	(* Tipologia di presa della falda *)
	TPICK_LAY_VENTOSE							:= 4,		(* Identifica la presa di tipo FALDA A VENTOSE, utilizzata nel pal. Lastre *)
	TPICK_LAY_ARPIONI							:= 5,		(* Identifica la presa di tipo FALDA CON ARPIONI, utilizzata nel pal. Lastre per il polistirolo *)
	
	TPICK_QUADROTTA								:= 10		(* Identifica la presa di tipo LASTRA (CLASSICA A VENTOSE) *)

	//TPICK_UNDEFINED								 := 99     
);
END_TYPE
//  TPICK_NOT_DEFINED = '-1'

// ---- Data types/Enum/e_Tipo_Traiettoria.TcTLEO
{attribute 'Tc2GvlVarNames'}
{attribute 'strict'}
(* Tipi Traiettoria *)
TYPE e_Tipo_Traiettoria :
(
	TRAIETTORIA_SENZA_APPROCCIO	:= 0,	(* Identifica che il punto di approccio coincide con il punto di deposito *)
	TRAIETTORIA_CON_APPROCCIO	:= 1	(* Identifica che il punto di approccio dipende dai valori di Ax,Ay,Az della lastra in deposito *)
);
END_TYPE

// ---- Data types/Enum/e_Verso_Pallettizzatore.TcTLEO
{attribute 'Tc2GvlVarNames'}
{attribute 'strict'}
//Verso del Pallettizzatore
TYPE e_Verso_Pallettizzatore :
(
	PALLETTIZZATORE_DX := 1, //Identifica il pallettizzatore la cui linea di trasporti rimane ALLE SPALLE e A DESTRA
	PALLETTIZZATORE_SX := 2 //Identifica il pallettizzatore la cui linea di trasporti rimane ALLE SPALLE e A SINISTRA
);
END_TYPE

// ---- Data types/Enum/Formatura/e_TipologiaDeposito.TcDUT
{attribute 'Tc2GvlVarNames'}
{attribute 'strict'}
TYPE e_TipologiaDeposito :
(
	NOT_DEFINED				:= -1,
	ORIZZONTALE				:= 1,		// TIPO DI DEPOSITO ORIZZONTALE (CASSA E PALLET)
	INCLINATO				:= 2,		// TIPO DI DEPOSITO INCLINATO (CAVALLINA)
	INCLINATO_LATOSINGOLO	:= 3		// TIPO DI DEPOSITO INCLINATO CON UN SOLO LATO DI DEPOSITO (BUNDLE)
);
END_TYPE

// ---- Data types/Enum/Trasporti/e_ElementZone.TcDUT
{attribute 'Tc2GvlVarNames'}
{attribute 'strict'}
TYPE e_ElementZone :
(
	NULL				:= -1,
	RullCarico 			:= 0,
	RullCarico2 		:= 1,
	RullCentrIngresso 	:= 2,
	RullCentrIngresso2 	:= 3,
	RullMobile 			:= 4,
	RullMobile2 		:= 5,
	RullP1 				:= 6,
	RullP1_2 			:= 7,
	RullP2 				:= 8,
	RullP2_2 			:= 9,
	RullSC1 			:= 10,
	RullSC1_2 			:= 11,
	RullSC2 			:= 12,
	RullSC2_2 			:= 13	
	
);
END_TYPE

// ---- Data types/Enum/Trasporti/e_PosizioneRullieraMobile.TcDUT
{attribute 'Tc2GvlVarNames'}
//{attribute 'strict'}
TYPE e_PosizioneRullieraMobile :
(
	POSIZIONE_INDEFINITA 	:= 0, 	//Posizione Indefinita
	POSIZIONE_CARICO 		:= 1,	//Posizione Rulliera Carico
	POSIZIONE_SCARICO 		:= 2,	//Posizione Rulliera Scarico
	POSIZIONE_RP1 			:= 3,	//Posizione Rulliera Prelievo 1
	POSIZIONE_RP2 			:= 4,	//Posizione Rulliera Prelievo 2
	POSIZIONE_ATTUALE 		:= 5	//Posizione Rulliera ATTUALE, NON SI CAMBIA LA DESTINAZIONE!
);
END_TYPE

// ---- Data types/Enum/Trasporti/e_StatoCentratura.TcDUT
{attribute 'Tc2GvlVarNames'}
{attribute 'strict'}
TYPE e_StatoCentratura :
(
	CENTRATURA_DISABILITATA		:= 0, 
	CENTRATURA_DA_ESEGUIRE	:= 1, 
	CENTRATURA_ESEGUITA 		:= 2
);
END_TYPE

// ---- Data types/Enum/Trasporti/e_TipoMacchinaTrasporti.TcDUT
{attribute 'Tc2GvlVarNames'}
{attribute 'strict'}
TYPE e_TipoMacchinaTrasporti :
(
	Macchina_ZonaPal := 0,//Zona Pallettizzatore
	Macchina_ZonaBS := 1 //Zona BAnco Scelta
);
END_TYPE

// ---- Data types/LGV/e_Tipo_Richiesta_LGV.TcTLEO
{attribute 'Tc2GvlVarNames'}
{attribute 'strict'}
//Tipo Richiesta LGV
TYPE e_Tipo_Richiesta_LGV :
(
	REQ_PRELIEVO_LGV_PIENO	:= 1,	(* Tipo di richiesta LGV = Richiesta di Tipo "PRELIEVO DI ELEMENTO CON MATERIALE" *)
	REQ_DEPOSITO_LGV_PIENO	:= 2,	(* Tipo di richiesta LGV = Richiesta di Tipo "DEPOSITO ELEMENTO CON MATERIALE" *)
	REQ_PRELIEVO_LGV_VUOTO	:= 3,	(* Tipo di richiesta LGV = Richiesta di Tipo "PRELIEVO ELEMENTO SENZA MATERIALE" *)
	REQ_DEPOSITO_LGV_VUOTO	:= 4	(* Tipo di richiesta LGV = Richiesta di Tipo "DEPOSITO ELEMENTO SENZA MATERIALE" *)
	
);
END_TYPE

// ---- Data types/LGV/e_Stato_Richiesta_LGV_1.TcTLEO
{attribute 'Tc2GvlVarNames'}
{attribute 'strict'}
//Stato Richiesta LGV
TYPE e_Stato_Richiesta_LGV_1 :
(
	NESSUNA_REQ_LGV	 	:= 0,	(* NESSUNA RICHIESTA/CHIAMATA LGV *)
	REQ_LGV			 	:= 1 	(* CHIAMATA LGV *)
);
END_TYPE

// ---- Data types/LGV/LGV_Stato_Formatura.TcDUT
TYPE LGV_Stato_Formatura :
STRUCT

CodicePallet 	: INT; //Codice del Pallet Presente in formatura
CodiceFalda		: INT; //Codice della Falda presente in formatura
PacchiPresenti_ZonaPositiva : INT; //Numero dei pacchi presenti della formatura nella zona Positiva(rispetto al ribaltino)
PacchiPresenti_ZonaNegativa : INT; //Numero dei pacchi presenti della formatura nella zona Negativa(rispetto al ribaltino)

END_STRUCT
END_TYPE

// ---- Data types/LGV/LGV_Stato_Pallettizzatore.TcDUT
TYPE LGV_Stato_Pallettizzatore :
STRUCT
	(* Stato del Pallettizzatore *)
	Automatico 	: BOOL; //Identifica lo stato di AUTOMATICO del Pallettizzatore
	Errore 		: BOOL; //Identifica lo stato di ERRORE del Pallettizzatore

END_STRUCT
END_TYPE

// ---- Data types/LGV/LGV_Stato_Postazione.TcDUT
TYPE LGV_Stato_Postazione :
STRUCT

	Abilitata			: INT; 	 // Abilitazione: 0=Postazione DISABILITATA, 1=Postazione ABILITATA
	Tipologia 			: INT; 	 // Tipologia: 1=Catasta Vuoti, 2=Pallet Singolo, 3=Falda,
	ProgressiveNr 		: UDINT; //Ad ogni deposito PALLET viene incrementato il suo valore ("ID univoco del pallet depositato")
	LGV_Req 			: INT; 	 //Chiamata Navetta: 0=Nessuna Chiamata, 1=Chiamata LGV
	CodicePallet 		: INT;	 //Codice identificativo del Pallet
	CodiceFalda 		: INT;	 //Codice identificativo della Falda
	CodiceLavorazione 	: INT;	 //Codice identificativo di lavorazione 
	AltezzaPallet		: REAL;	 //Altezza REALE degli elemti sulla Postazione
	
	Stato 				: INT; 	//Stato della Postazione
	CodiceFormatura 	: INT; 	//Codice di Formatura Associata alla postazione
	NPaccoSuccesivo 	: INT;	//Numero del pacco da depositare
	PN					: INT;	//Quota X postazione rispetto all quota X del ribaltino (0=Positiva, 1=Negativa)
	LGVAttr				: INT;   //Identifica gli attributi che il pallet completo dovrà avere (Tipo di Nastratura,avvolgitura,ecc)

END_STRUCT
END_TYPE

// ---- Data types/LGV/e_Stato_Operazione_LGV.TcTLEO
{attribute 'Tc2GvlVarNames'}
{attribute 'strict'}
//Stato Operazione LGV
TYPE e_Stato_Operazione_LGV :
(
	LGV_OPERAZIONE_VERIFICATA 	:= 0,	(* Indica che l'operazione svolta da parte del veicolo è stata verificata *)
	LGV_PRELIEVO_EFFETTUATO 	:= 1,	(* Indica che il prelievo da parte del veicolo è stato effettuato *)   
	LGV_DEPOSITO_EFFETTUATO 	:= 2	(* Indica che il deposito da parte del veicolo è stato effettuato *)
);
END_TYPE

// ---- Data types/Nuove/ST_OffsetAllDirection.TcDUT
TYPE ST_OffsetAllDirection :
STRUCT
	X90 : REAL := 0.0;	(* (mm) OFFSET di deposito direzione X, utilizzato per PALLET o CASSE *)
	Y90 : REAL := 0.0;	(* (mm) OFFSET di deposito direzione Y, utilizzato per PALLET o CASSE *)
	Z90 : REAL := 0.0;	(* (mm) OFFSET di deposito direzione Z, utilizzato per PALLET o CASSE *)
	J90 : REAL := 0.0;	(* (mm) OFFSET di deposito direzione J, utilizzato per PALLET o CASSE *)
	
	X0 	: REAL := 0.0;	(* (mm) OFFSET di deposito direzione X, utilizzato per CAVALLETTI *)
	Y0 	: REAL := 0.0;	(* (mm) OFFSET di deposito direzione Y, utilizzato per CAVALLETTI *)
	Z0 	: REAL := 0.0;	(* (mm) OFFSET di deposito direzione Z, utilizzato per CAVALLETTI *)
	J0 	: REAL := 0.0;	(* (mm) OFFSET di deposito direzione J, utilizzato per CAVALLETTI *)
	
	X180 : REAL := 0.0;	(* (mm) OFFSET di deposito direzione X, utilizzato per CAVALLETTI *)
	Y180 : REAL := 0.0;	(* (mm) OFFSET di deposito direzione Y, utilizzato per CAVALLETTI *)
	Z180 : REAL := 0.0;	(* (mm) OFFSET di deposito direzione Z, utilizzato per CAVALLETTI *)
	J180 : REAL := 0.0;	(* (mm) OFFSET di deposito direzione J, utilizzato per CAVALLETTI *)

END_STRUCT
END_TYPE

// ---- Data types/Nuove/TFMachinePalletizer_ListaProduzione_WAM_HMI.TcDUT
TYPE TFMachinePalletizer_ListaProduzione_WAM_HMI :
STRUCT
	Stato					: INT		:= -1;	(* Stato Elemento *)
	Support					: TFMachinePalletizer_Pallet; (* Tipologia supporto *)
	PElementList			: ARRAY [1..MAXELEMENTLIST] OF TFMachinePalletizer_PlaceElementList ; (* Elemento Da Movimentare *)
	NumeroListaAssociata 	: UINT := 0;//Indica il numero della lista associata a questa postazione nel caso ci siano + liste possibili es. post 1-4/5-8..																								
END_STRUCT
END_TYPE

// ---- Data types/Nuove/TFMachinePalletizer_WorkAreaTransport_State.TcDUT
TYPE TFMachinePalletizer_WorkAreaTransport_State :
STRUCT
	
	IDElement 		: UDINT; //ID univoco generato dalla macchina  per il tracking degli alementi
	
	State			: e_Stato_PickPoint	:= 0;	(* Stato della rulliera (0=Rulliera In Manuale, 1=Rulliera in Automatico, 2=Rulliera in Allarme *)
	PowerOK			: BOOL  := FALSE; (* Indica che ho la marcia degli ausiliari delle rulliere *)
	ProdPresence	: e_Stato_Prodotto_Generico	:= PROD_ASSENTE;	(* Stato di Presenza prodotto (0=Prodotto Assente, 1=Prodotto Presente *)
	ReadyToWork		: BOOL  := 0;	(* Indica che si puù lavorare sul supporto, quindi prelevare o depositare elementi *)
	Priority		: INT   := 0;	(* Priorità del punto di prelievo, Attualmente: 0 = Priorità MINIMA, 1 = Priorità MASSIMA *)
	
	Element			: TFMachinePalletizer_PlaceElement; (* Struttura Usata per Tracciare l'elemento presente *)
	DataElement		: TFMachinePalletizer_DataElement; (* Struttura dati che la macchina acquisisce/trasferisce in fase di pallettizzazione/depallettizazione *)
	Supporto		: TFMachinePalletizer_Pallet; (* Struttura del supporto presente sul punto di prelievo *)
	
	StatoPrelievo	: INT   := 0;	(* WRITE - Stato del prelievo: 0 = Da effettuare, 1 = Effettuato *)		
	StatoIngombroEE	: INT   := 0;	(* WRITE - Stato dell'ingombro dell'End-Effector: 0 = Non in ingombro, 1 = In Ingombro *)	
	
	XPosBandella		: REAL  := 0.0; (* Quota Bandella, Scritta dalle Rulliere (se posizionamento motorizzato) oppure dall'operatore (misura dal punto fiso della rulliera alla bandella) *)
	YPosBandella		: REAL  := 0.0; (* Quota Bandella, Scritta dalle Rulliere (se posizionamento motorizzato) oppure dall'operatore (misura dal punto fiso della rulliera alla bandella) *)
	
	NumeroPrelDepEffettuati : UINT := 0; (* Numero prelievi/Depositi effettuati sulle'elemento attuale *)
	
END_STRUCT
END_TYPE

// ---- Data types/Nuove/TFMachinePalletizer_WorkPlacePointToPalletizer.TcDUT
TYPE TFMachinePalletizer_WorkPlacePointToPalletizer :
STRUCT

	State					: e_Stato_PickPoint	:= 0;	(* Stato della rulliera (0=Rulliera In Manuale, 1=Rulliera in Automatico, 2=Rulliera in Allarme *)
                         
	PhaseStopDone 			: BOOL;(*Richiesta Stop in fase ESEGUITA*)
                            
	IDElement 				: UDINT; (*ID univoco generato dalla macchina  per il tracking degli alementi*)
	SupportPresent 		 	: BOOL;(* Supporto presente sul punto di deposito e pronto per essere pallettizzato *) 	
	Support 				: TFMachinePalletizer_Pallet; (* Struttura del supporto presente sul punto di prelievo *)
		
END_STRUCT
END_TYPE

// ---- Data types/Nuove/TFMachinePalletizer_WorkPlacePointFromPalletizer.TcDUT
TYPE TFMachinePalletizer_WorkPlacePointFromPalletizer :
STRUCT

	PhaseStopReq 			: BOOL;(*Richiesta Stop in fase*)
                            
	SupportREQ 				: BOOL;(* Richiesta del supporto punto di depostio *)
	Support				  	: TFMachinePalletizer_Pallet;(* Struttura del supporto richiesto sul punto di deposito *)
                                                 
	StatoIngombroEE			: INT   := 0;	(* Stato dell'ingombro dell'End-Effector: 0 = Non in ingombro, 1 = In Ingombro *)	
	
	ElementCompleted		: BOOL; (* Indica che l'elemento è stato completato *)

	State					: INT;//STtao pallettizzatore

	NextSupport			  	: TFMachinePalletizer_Pallet;(* Struttura del supporto successivo richiesto sul punto di deposito *)
   
END_STRUCT
END_TYPE

// ---- Data types/Picking/e_TypologySupDataPicking.TcDUT
{attribute 'strict'}
TYPE e_TypologySupDataPicking :
(
	//0= Orrizzontale LEGNO,1= Orrizzontale Telaio , 2 = Bundle, 3 = A-FRAME
	LEGNO_PIANO 	:= 0, //Legno/Pallet in piano
	TELAIO_PIANO 	:= 1, //Telaio in ferro in piano
	BUNDLE_VERT 			:= 2, //Bundle posteriore
	A_FRAME_VERT 		:= 3 //A-FRAME 
);
END_TYPE

// ---- Data types/Picking/ST_DataManualPicking.TcDUT
TYPE ST_DataManualPicking :
STRUCT
	ID_LIST			: STRING(255) 	:= '';	(* Identificatore univoco della LISTA da Eseguire *)
	State			: INT			:= -1;	(*Stato della lista in lavoro *)
	SlabNumber  	: UINT 			:= 0; (* Numero di lastre da depositare sul supporto *)
	SlabDimension 	: TFDimensionElement; (* Dimensione Lastra *)
	Layer 			: ST_LayerData; (* Struttura descrizione falda *)
	LayerSequence 	: INT; (* Sequenza di deposito delle falde -> 0=Nessuna falda,1=Deposito dopo ogni lastra,2=Deposito ogni 2 lastre,ecc*)
	SupportPianoLegno	: ST_SupportData; (* Dati del supporto in piano per legni*)
	SupportPianoFerro	: ST_SupportData; (* Dati del supporto in piano per ferro*)
	SupportVertBundle	: ST_SupportData; (* Dati del supporto in verticale per bundle*)	
	SupportVertCav		: ST_SupportData; (* Dati del supporto in verticale per cavalletto*)	
END_STRUCT
END_TYPE

// ---- Data types/Picking/ST_WorkAreaDataPicking.TcDUT
TYPE ST_WorkAreaDataPicking :
STRUCT
	Destinazione		  		: BOOL;	//Se TRUE=WA di destinazione materiale, FALSE=Postazione di prelievo materiale
	NumElementiDaLavorare 		: UINT; 	//Numero elementi da depositare-prelevare
	Typology			  		: INT := 0; 	//Supporto disposto in verticale: e_TypologySupDataPicking: 0= Orrizzontale LEGNO,1= Orrizzontale Telaio , 2 = Bundle, 3 = A-FRAME 
	TipoTrabajoLado_Cavallete 	: INT := 0; // // 0-trabaja aambos lados 1-Lado 0 Grados 2-Lado 180 Grados
END_STRUCT
END_TYPE

// ---- Data types/Programmi Movimento/TFModulePortaleStatus.TcDUT
TYPE TFModulePortaleStatus :
STRUCT
	
	X				: ST_MachinePalletizerAxeState;	(* X Axe State (UI Position=mm, UI Velocity=mm/sec UI Acc/Dec=mm/sec2) *)
	Y				: ST_MachinePalletizerAxeState;	(* Y Axe State (UI Position=mm, UI Velocity=mm/sec UI Acc/Dec=mm/sec2) *)
	Z				: ST_MachinePalletizerAxeState;	(* Z Axe State (UI Position=mm, UI Velocity=mm/sec UI Acc/Dec=mm/sec2) *)
	J				: ST_MachinePalletizerAxeState;	(* J Axe State (UI Position=°,  UI Velocity=°/sec  UI Acc/Dec=°/sec2) *)
	K				: ST_MachinePalletizerAxeState;	(* K Axe State (UI Position=mm, UI Velocity=mm/sec UI Acc/Dec=mm/sec2) *)
	Pinza 			: ST_MachinePalletizerPinzaStateComplete; (* State Pinza *)
	
	Macchina   		: ST_MachinePalletizerMachineState; (* Stato del modulo di gestione Della Macchina *)

	ModAsse_X 		: ST_MachinePalletizerModuleState; (* Stato del modulo di gestione Asse X *)
	ModAsse_Y 		: ST_MachinePalletizerModuleState; (* Stato del modulo di gestione Asse Y *)
	ModAsse_Z 		: ST_MachinePalletizerModuleState; (* Stato del modulo di gestione Asse Z *)
	ModAsse_J 		: ST_MachinePalletizerModuleState; (* Stato del modulo di gestione Asse J *)
	ModAsse_K 		: ST_MachinePalletizerModuleState; (* Stato del modulo di gestione Asse K *)
	ModPinza 		: ST_MachinePalletizerModuleState; (* Stato del modulo di gestione Pinza *)
	ModLettoreBc 	: ST_MachinePalletizerModuleState; (* Stato del modulo di gestione Lettore Barcode *)
	
END_STRUCT
END_TYPE

// ---- Data types/StatoPostazioneHMI.TcDUT
TYPE StatoPostazioneHMI :
STRUCT

	Abilitata			: INT; 	 // Abilitazione: 0=Postazione DISABILITATA, 1=Postazione ABILITATA
	TipologiaPostazione	: INT; 	 // Tipologia: 1=Catasta Vuoti, 2=Pallet Singolo, 3=Falda,
	ProgressiveNr 		: UDINT; //Ad ogni deposito PALLET viene incrementato il suo valore ("ID univoco del pallet depositato")
	
	LGV_Req 			: INT; 	 //Chiamata Navetta: 0=Nessuna Chiamata, 1=Chiamata LGV
	TipologiaSupporto   : INT;
	CodiceLavorazione 	: INT;	 //Codice identificativo di lavorazione 
	
	Stato 				: INT; 	//Stato della Postazione
	CodiceFormatura 	: INT; 	//Codice di Formatura Associata alla postazione
	NPezzi			 	: INT;	//Numero dei pezzi presenti
	

END_STRUCT
END_TYPE

// ---- Data types/Nuove/TFCodiciPerFormatura.TcDUT
TYPE TFCodiciPerFormatura :
STRUCT
	Code : ARRAY[1..MAXFORMINGCODE] OF INT;
END_STRUCT
END_TYPE

// ---- Data types/Nuove/TFError_WAM.TcDUT
TYPE TFError_WAM :
STRUCT
	Code 		: UINT; (*Codice di errore*)
	ExtraCode 	: UINT; (*Codice di errore EXTRA*)
END_STRUCT
END_TYPE

// ---- Data types/Nuove/TFMachinePalletizer_DataElementMP.TcDUT
TYPE TFMachinePalletizer_DataElementMP :
STRUCT
	RequetsID 		: DINT	:= 0; (* Scheduler ID *)
	Article 			: STRING(49) := '';
	ArticleDescription 	: STRING(49) := '';(* Descrizione Articolo *)
	Tono			: STRING(19)	:= '';	(* Tono Elemento *)
	Scelta			: STRING(19)	:= '';	(* Scelta Elemento *)
	Calibro			: STRING(19)	:= '';	(* Calibro Elemento *)
	
	Lenght 		: INT := 0; //Lunghezza
	Width 		: INT := 0; //Larghezza
	Thickness 	: INT := 0; //Spessore
END_STRUCT
END_TYPE

// ---- Data types/Nuove/TFMachinePalletizer_PinzaVentoseManCmd.TcDUT
TYPE TFMachinePalletizer_PinzaVentoseManCmd :
STRUCT
	
	AttivazioneVuotoDX			: BOOL;//Attivazione vuoto Ovem DX 
	AttivazioneVuotoSX			: BOOL;//Attivazione vuoto Ovem SX

	DisattivazioneVuotoDX			: BOOL;//Comandi Ovem
	DisattivazioneVuotoSX			: BOOL;//Comandi Ove

	ApriPinza				: BOOL; //Apertura Pinza
	ChiudiPinza				: BOOL; //Apertura Pinza

	SbloccoPinza			: BOOL;//Sblocco rotazione
	BloccoPinza				: BOOL;//Blocco rotazione

	AttivazioneVuotoFaldeDX 	: BOOL;//Attivazione aspirazione Falde DX
	DisattivazioneVuotoFaldeDX	: BOOL;//Disattivazione aspirazione Falde DX
	
	AttivazioneVuotoFaldeSX 	: BOOL;//Attivazione aspirazione Falde SX
	DisattivazioneVuotoFaldeSX	: BOOL;//Disattivazione aspirazione Falde SX

	AttivaTastatori : BOOL; //Attivazione Tastatori
	DisattivaTastatori : BOOL; //Disattivazione Tastatori
	
	CalibrazioneOVEM : bool; //Calibrazione OVEM

END_STRUCT
END_TYPE

// ---- Data types/Nuove/TFMachinePalletizer_ApprendimentoQuota.TcDUT
TYPE TFMachinePalletizer_ApprendimentoQuota :
STRUCT
	Stato			: e_Stato_Apprendimento	:= e_Stato_Apprendimento.NOT_DEFINED;	(* Stato apprendimento Direzione X 0=Disabilitato, 1=Abilitato da Eseguire, 2=Eseguito, -1 dato non valido *)
	QuotaStart		: LREAL	:= 0.0;	(* (mm) Quota inizio Apprendimento Direzione X *)
	QuotaRilevata	: LREAL	:= 0.0; (* Quota rilevata durante apprendimento Direzione X *)
END_STRUCT
END_TYPE

// ---- Data types/Nuove/TFMachinePalletizer_CoordinateApprendimento.TcDUT
TYPE TFMachinePalletizer_CoordinateApprendimento :
STRUCT
	X : TFMachinePalletizer_LatoApprendimento;
	Y : TFMachinePalletizer_LatoApprendimento;
	Z : TFMachinePalletizer_LatoApprendimento;
	J : TFMachinePalletizer_LatoApprendimento;
END_STRUCT
END_TYPE

// ---- Data types/Nuove/TFMachinePalletizer_LatoApprendimento.TcDUT
TYPE TFMachinePalletizer_LatoApprendimento :
STRUCT
	Lato0 	: TFMachinePalletizer_ApprendimentoQuota;	
	Lato90 	: TFMachinePalletizer_ApprendimentoQuota;
	Lato180 : TFMachinePalletizer_ApprendimentoQuota;
END_STRUCT
END_TYPE

// ---- Data types/Nuove/TFMachinePalletizer_DataElement.TcDUT
TYPE TFMachinePalletizer_DataElement :
STRUCT
	WorkingID 			: STRING	:= ''; (* Identifica l'ID univoco della lavorazione da eseguire *)
	
	Codice				: STRING	:= '';	(* Codice Elemento *)
	Scelta				: STRING	:= '';	(* Scelta Elemento *)
	Tono				: STRING	:= '';	(* Tono Elemento *)
	Calibro				: STRING	:= '';	(* Calibro Elemento *)
	Quantity  			: UINT 		:= 0;	(* Quantità *)
	ArticleDescription 	: STRING(50) := '';(* Descrizione Articolo *)
END_STRUCT
END_TYPE

// ---- Data types/Nuove/TFMachinePalletizer_EndEffector.TcDUT
TYPE TFMachinePalletizer_EndEffector :
STRUCT
	Tipologia 	: INT := -1; 	//Indica la tipologia dell'elemento 
	Lunghezza 	: REAL := 0; 	//Indica la lunghezza dell'elemento
	Larghezza 	: REAL := 0; 	//Indica la larghezza dell'elemento	
	Spessore	: REAL := 0; 	//Indica lo spessore dell'elemento
	PosizioneBC_X : REAL := 0;	//Indica la posizione del barcode lungo la sua lunghezza e rispetto il punto medio
	PosizioneBC_Y : REAL := 0;	//Indica la posizione del barcode lungo la sua larghezza e rispetto il punto medio	
	PosizioneBC_Z : REAL := 0;	//Indica la posizione del barcode lungo il suo spessore e rispetto il punto medio
END_STRUCT
END_TYPE

// ---- Data types/Nuove/TFMachinePalletizer_BarCode.TcDUT
TYPE TFMachinePalletizer_BarCode :
STRUCT
	State 	: e_Stato_LetturaBarCode := LETURA_BC_TERMINATA;				(* Identifica lo stato della Lettura del BC:	0= Non Ancora letto/Da Leggere, 
																					1= Lettura In corso
																					2= Codice Letto e Valido/Non da leggere, 
																					3= Errore *)
	ErrorCode	: INT := 0;				(* Identifica il codice di errore *)
	Value		: STRING[DIMBARCODE];	(* Identifica il valore della lettura *)	
END_STRUCT
END_TYPE

// ---- Data types/Nuove/TFMachinePalletizer_ListaProduzione.TcDUT
TYPE TFMachinePalletizer_ListaProduzione :
STRUCT
	ID_LIST		: STRING(255) 					:= '';	(* Identificatore univoco della LISTA da Eseguire *)
	State		: e_Stato_ListaDiProduzione		:= -1;	(*Stato della lista in lavoro *)
	SlabNumber  : UINT := 0; (* Numero di lastre da depositare sul supporto *)
	SlabData 	: ARRAY[1..MAXARTICLEPICKING] OF TFMachinePalletizer_DataElement; (* Lastra che serve per comporre l'ordine finale, ordinato in base alla sequenza richiesta 1=Primo prodotto da pallettizzare *)
	SlabDimension 	: TFDimensionElement; (* Dimensione Lastra *)
	LayerSequence 	: UINT := 0;//Sequenza di deposito delle falde -> 0=Nessuna falda,1=Deposito dopo ogni lastra,2=Deposito ogni 2 lastre,ecc
	LayerCode     	: UDINT := 0; (* Codice della falda da deposotare *)
	Support			: UDINT := 0; (* Codice pallet su cui eseguire la pallettizzazione *)
											
END_STRUCT
END_TYPE

// ---- Data types/Nuove/TFMachinePalletizer_ListaProduzione_WAM.TcDUT
TYPE TFMachinePalletizer_ListaProduzione_WAM :
STRUCT
	Stato					: e_Stato_ListaDiProduzione		:= -1;	(* Stato Elemento *)
	Support					: TFMachinePalletizer_Pallet; (* Tipologia supporto *)
	PElementList			: ARRAY [1..MAXELEMENTLIST] OF TFMachinePalletizer_PlaceElementList ; (* Elemento Da Movimentare *)
	Forming 				: TFMachinePalletizer_FormingForSlab;
	NumeroListaAssociata 	: UINT := 0;//Indica il numero della lista associata a questa postazione nel caso ci siano + liste possibili es. post 1-4/5-8..												
END_STRUCT
END_TYPE

// ---- Data types/Nuove/TFMachinePalletizer_OffsetElement.TcDUT
TYPE TFMachinePalletizer_OffsetElement :
STRUCT
	Dir_X 				: REAL := 0.0;	(* (mm) OFFSET in direzione X *)
	Dir_Y 				: REAL := 0.0;	(* (mm) OFFSET in direzione Y (+ è grande + mi allontano dal supporto)*)
	Dir_Z 				: REAL := 0.0;	(* (mm) OFFSET in direzione Z (+ è grande + mi allontano dal supporto)*)
	Dir_J 				: REAL := 0.0;	(* (°) OFFSET di inclinazione J (Pinza Inclinata: + è grande + è grande l'inclinazione, 
																		Pinza Pari: più è grande più si sposta verso l'angolo maggiore *)
	
END_STRUCT
END_TYPE

// ---- Data types/Nuove/TFMachinePalletizer_PickPlaceParameters.TcDUT
TYPE TFMachinePalletizer_PickPlaceParameters :
STRUCT

	OffsetZPlaceLayer			: REAL;	(* Offset quota Z per rilascio falda *)
			
	XPickApproach	: LREAL	:= 100.0;		(* (mm) Offset di Approccio X in prelievo *)
	YPickApproach	: LREAL	:= 100.0;		(* (mm) Offset di Approccio Y in prelievo *)
	ZPickApproach	: LREAL	:= 100.0;		(* (mm) Offset di Approccio Z in prelievo *)
	JPickApproach	: LREAL	:= 100.0;		(* (mm) Offset di Approccio J in prelievo *)
	//KPickApproach	: LREAL	:= 0.0;		(* (mm) Offset di Approccio in prelievo *)
	//WPickApproach	: LREAL	:= 0.0;		(* (mm) Offset di Approccio in prelievo *)
	
	XPlaceApproach	: LREAL	:= 100.0;		(* (mm) Offset di Approccio X in deposito *)
	YPlaceApproach	: LREAL	:= 100.0;		(* (mm) Offset di Approccio Y in deposito *)
	ZPlaceApproach	: LREAL	:= 100.0;		(* (mm) Offset di Approccio Z in deposito *)
	JPlaceApproach	: LREAL	:= 100.0;		(* (mm) Offset di Approccio in deposito *)
	//KPlaceApproach	: LREAL	:= 0.0;		(* (mm) Punto di Approccio in deposito *)
	//WPlaceApproach	: LREAL	:= 0.0;		(* (mm) Punto di Approccio in deposito  *)

END_STRUCT
END_TYPE

// ---- Data types/Nuove/TFMachinePalletizer_PinzaState.TcDUT
TYPE TFMachinePalletizer_PinzaState :
STRUCT
	LatoDxAperto : BOOL; //Indica che la prolunga DX della pinza è aperta
	LatoSxAperto : BOOL; //Indica che la prolunga SX della pinza è aperta
	LatoDxChiuso : BOOL; //Indica che la prolunga DX della pinza è chiusa
	LatoSxChiuso : BOOL; //Indica che la prolunga SX della pinza è chiusa
	
	LatoSxPiastrellaInPresa : BOOL; //Indica che sul lato SX ho in presa la piastrella
	LatoDxPiastrellaInPresa : BOOL; //Indica che sul lato DX ho in presa la piastrella

	LatoSxFaldaInPresa 		: BOOL; //Indica che sul lato SX ho in presa la FALDA
	LatoDxFaldaInPresa 		: BOOL; //Indica che sul lato DX ho in presa la FALDA
	
	RotazioneSbloccata 	: BOOL; //Indica che la Rotazione lungo z è sbloccata
	RotazioneBloccata	: BOOL; //Indica che la rotazione lungo z è bloccata
	
	ElementoPrelevato : BOOL;//Indica che l'elemento è stato prelevato
	
	LetturaFTC0 	: REAL;
	LetturaFTC180 	: REAL;
	
	LetturaFTC0_2 	: REAL;
	LetturaFTC180_2 : REAL;
	
	PianoInPresa : BOOL;
END_STRUCT
END_TYPE

// ---- Data types/Nuove/TFMAchinePalletizer_PinzaVentoseStatus.TcDUT
TYPE TFMAchinePalletizer_PinzaVentoseStatus :
STRUCT

	Module : TFMachinePalletizer_ModuleState;

	CilindroApertura 			: TF_CylinderState;
	CilindroSbloccoRotazione 	: TF_CylinderState;
	AspirazioneFaldaDX 			: TF_CylinderState;
	AspirazioneFaldaSX 			: TF_CylinderState;
	AspirazioneDX 				: TF_CylinderState;
	AspirazioneSX 				: TF_CylinderState;		
	CilindroTasteggio			: TF_CylinderState;	
	AspirazioneDX2 				: TF_CylinderState;
	AspirazioneSX2 				: TF_CylinderState;		
	CilindroSbloccoBascolante 	: TF_CylinderState;
END_STRUCT
END_TYPE

// ---- Data types/Nuove/TFMachinePalletizer_PinzaVentose_OUT.TcDUT
TYPE TFMachinePalletizer_PinzaVentose_OUT :
STRUCT
END_STRUCT
END_TYPE

// ---- Data types/Nuove/TFMachinePalletizer_PlaceElement.TcDUT
TYPE TFMachinePalletizer_PlaceElement :
STRUCT
	(* Tipologia *)
	Typology		: e_Tipo_Elemento_Da_Lavorare := TERMINATORE;	(* Tipo di ELEMENTO DA LAVORARE: 0: LASTRA,1:FALDA *)
	TypologyCode	: INT						:= -1;	(* Descrittore tipo elemento *)
	(*Dimensione Lastra*) // Añadido Alberto 14-10-2025
	SlabDimension 								: TFDimensionElement; (* Dimensione Lastra *)
	DimensionPiezasLadoALadoB					: ES_dimensionPiezaLadoA_ladoB; 
	(* Dimensioni *)
	XDim		: REAL							:= 0.0;	(* (mm) Dimensione X *)
	YDim		: REAL							:= 0.0;	(* (mm) Dimensione Y *)
	ZDim		: REAL							:= 0.0;	(* (mm) Dimensione Z *)
	(* Quote di deposito *)
	X			: LREAL							:= 0.0;	(* (mm) Destination - Coordinata X *)
	Y			: LREAL							:= 0.0;	(* (mm) Destination - Coordinata Y *)
	Z			: LREAL							:= 0.0;	(* (mm) Destination - Coordinata Z *)
	J			: LREAL							:= 0.0;	(* (°)  Destination - Coordinata J (PITCH)*)
	CooCavallete : Es_CoordenadasCaballeteLadoA_ladoB  ;
	//K			: LREAL							:= 0.0;	(* (°)  Destination - Coordinata K (ROLL)*)
	//W			: LREAL							:= 0.0;	(* (°)  Destination - Coordinata W (YAW)*)

	(* Distanza di Accostamento *)
	AX			: REAL							:= 0.0; (* (mm) Approach X Distance - Distanza Accostamento X *)
	AY			: REAL							:= 0.0; (* (mm) Approach Y Distance - Distanza Accostamento Y *)
	AZ			: REAL							:= 0.0; (* (mm) Approach Z Distance - Distanza Accostamento Z *)
	AJ			: REAL							:= 0.0; (* (mm) Approach J Distance - Distanza Accostamento J (PITCH)*)
	//NUOVE???
	//AK			: REAL						:= 0.0; (* (mm) Approach Z Distance - Distanza Accostamento K (ROLL)*)
	//AW			: REAL						:= 0.0; (* (mm) Approach J Distance - Distanza Accostamento W (YAW)*)
	(* traiettoria di deposito *)
	Trajectory	: e_Tipo_Traiettoria			:= 0;	(* READ	- Tipo di percorso (0, 1, 2, 3, …) (-1 dato non valido) *)
	Empty : BOOL;//Indica che è vuoto
END_STRUCT
END_TYPE

// ---- Data types/Nuove/TFMachinePalletizer_PlaceElementList.TcDUT
TYPE TFMachinePalletizer_PlaceElementList :
STRUCT
	
	Stato 			: e_Stato_ElementoLista; (* Stato dell'elemento della lista*)
	
	PElement 		: TFMachinePalletizer_PlaceElement; (* Elemento Da Movimentare *)
	SlabData     	: TFMachinePalletizer_DataElement; (* Dati Elemento da depositare*)

	WA_PRELIEVO		: UINT	:= 0;	(* WA DOVE VIENE FATTO IL PRELIEVO *)
	WA_DEPOSITO		: UINT	:= 0;	(* WA DOVE VIENE FATTO IL DEPOSITO *)
	PP_PRELIEVO     : UINT	:= 0;	(* PICK-POINT DOVE VIENE FATTO IL PRELIEVO *)	
	
	Pareggiatura    : e_Stato_Pareggiatura_Lastra  := PAREGGIATURA_DISABILITATA;	(* Pareggiatura Lastra da eseguire Prima del deposito 0:NON ESEGUIRE, 1: DA ESEGUIRE, 2:ESEGUITA *)
	
END_STRUCT
END_TYPE

// ---- Data types/Nuove/TFMachinePalletizer_WorkPickPointOffset.TcDUT
TYPE TFMachinePalletizer_WorkPickPointOffset :
STRUCT
	X	:	REAL := 0.0; (* READ	- (mm) Offset del punto di prelievo in direzione X *)
	Y	:	REAL := 0.0; (* READ	- (mm) Offset del punto di prelievo in direzione Y *)
	Z	:	REAL := 0.0; (* READ	- (mm) Offset del punto di prelievo in direzione Z *)
	J	:	REAL := 0.0; (* READ	- (mm) Offset di rotazione del piano J *)
END_STRUCT
END_TYPE

// ---- Data types/Nuove/TFMachinePalletizer_WorkPickPoint_State.TcDUT
TYPE TFMachinePalletizer_WorkPickPoint_State :
STRUCT
	
	State			: INT	:= 0;	(* Stato della rulliera (0=Rulliera In Manuale, 1=Rulliera in Automatico, 2=Rulliera in Allarme *)
	PowerOK			: BOOL  := FALSE; (* Indica che ho la marcia degli ausiliari delle rulliere *)
	ProdPresence	: INT	:= 0;	(* Stato di Presenza prodotto (0=Prodotto Assente, 1=Prodotto Presente *)
	LastraPronta	: BOOL  := 0;	(* Indica che la lastra è pronta per essere prelevata *)
	Code			: INT	:= 0;	(* Codice Elemento *)
	Priority		: INT   := 0;	(* Priorità del punto di prelievo, Attualmente: 0 = Priorità MINIMA, 1 = Priorità MASSIMA *)
	
	Element			: TFMachinePalletizer_PlaceElement; (* Struttura Usata per Tracciare l'elemento presente *)

	StatoPrelievo	: INT   := 0;	(* WRITE - Stato del prelievo: 0 = Da effettuare, 1 = Effettuato *)		
	StatoIngombroEE	: INT   := 0;	(* WRITE - Stato dell'ingombro dell'End-Effector: 0 = Non in ingombro, 1 = In Ingombro *)	
	
	XPosBandella		: REAL  := 0.0; (* Quota Bandella, Scritta dalle Rulliere (se posizionamento motorizzato) oppure dall'operatore (misura dal punto fiso della rulliera alla bandella) *)
	YPosBandella		: REAL  := 0.0; (* Quota Bandella, Scritta dalle Rulliere (se posizionamento motorizzato) oppure dall'operatore (misura dal punto fiso della rulliera alla bandella) *)
	
	DataElement		: TFMachinePalletizer_DataElement; (* Struttura dati che la macchina acquisisce/trasferisce in fase di pallettizzazione/depallettizazione *)
		
END_STRUCT
END_TYPE

// ---- Data types/Nuove/TFMachinePalletizer_WorkPickPointRoller_State_DaLinea.TcDUT
TYPE TFMachinePalletizer_WorkPickPointRoller_State_DaLinea :
STRUCT
	
	Automatico		: BOOL	:= FALSE;	(* Stato della rulliera (FALSE=Rulliera In Manuale, TRUE=Rulliera in Automatico *)
	Errore			: BOOL	:= FALSE;	(* Stato della rulliera (FALSE=Rulliera senza Errori, TRUE=Rulliera in Errore *)
	PowerOK			: BOOL	:= FALSE;	(* Presenza Marcia (FALSE=Marcia Assente, TRUE=Marcia Presente *)
	Codice			: INT	:= 0;		(* Codice Prodotto *)
	Occupato		: BOOL  := FALSE;	(* Rulliera Occupata *)
	LastraPronta	: BOOL  := FALSE;	(* Lastra pronta e in posizione per prelievo *)
	Priority		: BOOL	:= FALSE;	(* Se true a parità di occupazione rispetto agli altri PickPoint, questo PickPoint ha la precedenza nel prelievo *)
	
END_STRUCT
END_TYPE

// ---- Data types/Nuove/TFMachinePalletizer_WorkPickPointRoller_State_ALinea.TcDUT
TYPE TFMachinePalletizer_WorkPickPointRoller_State_ALinea :
STRUCT
	
	Automatico			: BOOL 	:= FALSE;	(* Stato della rulliera (FALSE=Rulliera In Manuale, TRUE=Rulliera in Automatico *)
	PowerOK				: BOOL 	:= FALSE; 	(* Presenza Marcia (FALSE=Marcia Assente, TRUE=Marcia Presente *)
	Ingombro			: BOOL	:= FALSE;	(* Stato della rulliera (FALSE=Rulliera In Manuale, TRUE=Rulliera in Automatico *)
	Prelievo_Effettuato	: BOOL	:= FALSE ;	(* Se TRUE il prelievo è stato effettuato *)
	
END_STRUCT
END_TYPE

// ---- Data types/Nuove/TFMachinePalletizer_WorkPickPointStore_State.TcDUT
TYPE TFMachinePalletizer_WorkPickPointStore_State :
STRUCT
	
	ProdPresence	: INT	:= 0;	(* Stato PickPoint (0=Prodotto Assente, 1=Prodotto Presente *)
	Code			: INT   := -1;	(* Indica il codice della falda *)
		
	XDim			: REAL	:= 0;		(* (mm) Dimensione X Prodotto *)
	YDim			: REAL	:= 0;		(* (mm) Dimensione Y Prodotto *)
	ZDim			: REAL	:= 0;		(* (mm) Dimensione Z Prodotto *)
	
END_STRUCT
END_TYPE

// ---- Data types/Nuove/TFMachinePalletizer_WorkPickPointSlab.TcDUT
TYPE TFMachinePalletizer_WorkPickPointSlab :
STRUCT
	
	Tipologia			: e_Tipo_PickPoint 	:= -1;		(* Tipologia del punto di prelievo 
														Per lastre 	= RULLIERA;
														Per Falde	= MAGAZZIONO_FALDE *)
														
	ID					: INT 	:= -1;		(* Identifica il numero del PickPoint *)
	Enable				: INT	:= -1;		(* PickPoint Abilitata 0=no, 1=si, -1 dato non valido *)	
(***********************************************************************************************************************************************)
	X					: LREAL	:= 0.0;		(* (mm) Quota assoluta di impianto DA ORIGINE *)
	Y					: LREAL	:= 0.0;		(* (mm) Quota assoluta di impianto DA ORIGINE *)
	Z					: LREAL	:= 0.0;		(* (mm) Quota assoluta di impianto DA ORIGINE Caso di magazzino falde: è la quota della base di appoggio*)
	J					: LREAL	:= 0.0;		(* (mm) Quota assoluta di impianto DA ORIGINE *)
	ZRaise				: REAL  := 0.0; 	(* (mm) Quota di salita per uscire dall'ingombro *)
	
	///Lunghezza			: REAL := 0.0;		(* (mm) Ingombro in Lunghezza "X" rispetto il suo centro *)
	//Larghezza			: REAL := 0.0;		(* (mm) Ingombro in Larghezza "Y" rispetto il suo centro *)
	//Altezza				: REAL := 0.0;		(* (mm) Ingombro in Altezza "Z" rispetto il suo centro *)
	
	DoLearn_Z			: e_Stato_Apprendimento	:= -1;	(* Stato apprendimento Direzione Z 0=Disabilitato, 1=Abilitato da Eseguire, 2=Eseguito, -1 dato non valido *)
	Learn_Z				: REAL	:= 0.0;	(* (mm) Quota inizio Apprendimento Direzione Z *)
	Learned_Z			: LREAL	:= 0.0; (* (mm) Quota rilevata durante apprendimento Direzione Z *)
			
END_STRUCT
END_TYPE

// ---- Data types/Nuove/TF_CylinderState.TcDUT
TYPE TF_CylinderState :
STRUCT
	Active : BOOL;
	Inactive : BOOL;
	Error : UDINT;
	SensorActive : BOOL;
	SensorInactive : BOOL;
	StatusToHMI	: uint; //0= Null; 1= Active ; 2= Inactive; 3= Idle; 9 = Error ; 
END_STRUCT
END_TYPE

// ---- Data types/Nuove/TFMchinePalletizer_PinzaVentose_IN.TcDUT
TYPE TFMchinePalletizer_PinzaVentose_IN :
STRUCT
	TastoreCartoneSX : BOOL; //Sensore Tastatore lato SX
	TastoreCartoneDX : BOOL; //Sensore Tastatore lato SX
	ExtraCorsaPinzaSganciata : BOOL; //Sensore Di sicurezza rotazione lungo Z
	
	InKeyence0_Byte0 : BYTE;
	InKeyence0_Byte1 : BYTE;
	InKeyence180_Byte0 : BYTE;
	InKeyence180_Byte1 : BYTE;
	
	InKeyence0_Byte0_2 : BYTE;
	InKeyence0_Byte1_2 : BYTE;
	InKeyence180_Byte0_2 : BYTE;
	InKeyence180_Byte1_2 : BYTE;

	ByPassSensoreVuoto : BOOL;
	RichiestaRicalibrazioneOvemEsterna : BOOL;//Richiesta calibrazione esterna da macchina
	
	FTC_FaldaDX : BOOL;
	FTC_FaldaSX : BOOL;
	
END_STRUCT
END_TYPE

// ---- Data types/Nuove/TFPalletizerModules.TcDUT
TYPE TFPalletizerModules :
STRUCT
	AX_X 	: TFModulePalletizer_Ax;
	AX_Y 	: TFModulePalletizer_Ax;
	AX_Z 	: TFModulePalletizer_Ax;
	//AX_K 	: TFModulePalletizer_Ax;
	AX_J 	: TFModulePalletizer_AxJ_Lastre;
	Pinza 	: TFModulePalletizer_Pinza;
	

END_STRUCT
END_TYPE

// ---- Data types/Programmi Movimento/AxHomingParameters.TcDUT
TYPE AxHomingParameters :
STRUCT
	TipoHoming : INT; //Tipologia di homing da eseguire
	InvertiDirezione : BOOL; //FALSE=Direzione NEgativa, TRUE=Direzione positiva
END_STRUCT
END_TYPE

// ---- Data types/Programmi Movimento/Ax_Palletizer_Basic_Parameters.TcDUT
TYPE Ax_Palletizer_Basic_Parameters :
STRUCT
	Vel 	: REAL;
	Acc 	: REAL;
	Dec 	: REAL;
	Jerk 	: REAL;
	Torque 	: REAL;
END_STRUCT
END_TYPE

// ---- Data types/Programmi Movimento/Ax_Palletizer_Nominal_Parameters.TcDUT
TYPE Ax_Palletizer_Nominal_Parameters :
STRUCT
	ReferenceVelocity 		: REAL := 0.0;
	MaximumAcceleration 	: REAL := 0.0;
	MaximumDeceleration 	: REAL := 0.0;
	DefaultJerk 			: REAL := 0.0;
	DefaultTorque 			: REAL := 100.0;
END_STRUCT
END_TYPE

// ---- Data types/Programmi Movimento/Enum Programmi/e_ProgrammiMovimentoX.TcTLEO
{attribute 'Tc2GvlVarNames'}
{attribute 'strict'}
TYPE e_ProgrammiMovimentoX :
(
	
	X_PosDiRiposo					:= 0,
	X_PosFuoriIngombroRiposo 			:= 6,

	X_PosPrelievoFalda					:= 51,
	X_PosDepositoSuCatastaFalda			:= 52,
	X_PosDepositoFalda					:= 53,
	X_PosFuoriIngombroVuotoFalda		:= 56,

	X_PosStartLentaPrelievoLastra 		:= 101,
	X_PosPrelievoInLentaLastra 			:= 102,
	X_PosDistaccoLastraInLentaLastra	:= 103,
	X_PosStartLentaDepositoLastra 		:= 104,
	X_PosDepositoInLentaLastra			:= 105,
	X_PosFuoriIngombroVuotoLastra		:= 106,
	X_PosFuoriIngombroCaricoLastra		:= 126,
	X_PosGiroPiezaTraCavallete			:= 127
);
END_TYPE

// ---- Data types/Programmi Movimento/Enum Programmi/e_ProgrammiMovimentoJ.TcTLEO
{attribute 'Tc2GvlVarNames'}
{attribute 'strict'}
TYPE e_ProgrammiMovimentoJ :
(
	
	J_PosDiRiposo						:= 0,
	J_PosFuoriIngombro					:= 6,

	J_PosPrelievoFalda					:= 10,
	J_PosDepositoFalda					:= 11,
	
	J_PosPrelievoLastra					:= 12,
	J_PosDepositoLastra					:= 13,
	J_PosStartApproccioPrelLastra		:= 14,
	J_PosSfogliatura					:= 15,
	
	J_PosStartDepLastra					:= 16,
	
	J_PosPostScarico					:= 17,

	J_PosFuoriIngombroPosAttuale		:= 18

	
);
END_TYPE

// ---- Data types/Programmi Movimento/Enum Programmi/e_ProgrammiMovimentoY.TcTLEO
{attribute 'Tc2GvlVarNames'}
{attribute 'strict'}
TYPE e_ProgrammiMovimentoY :
(
	
	Y_PosDiRiposo						:= 0,
	Y_PosFuoriIngombroRiposo 			:= 6,

	Y_PosPrelievoFalda					:= 51,
	Y_PosDepositoSuCatastaFalda			:= 52,
	Y_PosDepositoFalda					:= 53,
	//Y_PosDepositoInLentaFalda			:= 55,
	Y_PosFuoriIngombroVuotoFalda 		:= 56,
	Y_PosFuoriIngombroCaricoFalda		:= 66,

	Y_PosStartLentaPrelievoLastra 		:= 101,
	Y_PosPrelievoInLentaLastra 			:= 102,
	Y_PosDistaccoLastraInLentaLastra	:= 103,
	Y_PosStartLentaDepositoLastra 		:= 104,
	Y_PosDepositoInLentaLastra			:= 105,
	Y_PosFuoriIngombroVuotoLastra		:= 106,
	Y_PosFuoriIngombroCaricoLastra		:= 126,
	Y_PosgiroPieza						:= 127,
	Y_PosPasillo0grados					:= 128,
	Y_PosPasillo180grados				:= 129
);
END_TYPE

// ---- Data types/Programmi Movimento/Enum Programmi/e_ProgrammiMovimentoZ.TcTLEO
{attribute 'Tc2GvlVarNames'}
{attribute 'strict'}
TYPE e_ProgrammiMovimentoZ :
(
	
	Z_PosDiRiposo						:= 0,
	Z_PosFuoriIngombroRiposo 			:= 6,

	Z_PosStartLentaPrelievoFalda		:= 51,
	Z_PosPrelievoInLentaFalda 			:= 52,
	Z_PosAttesaCadutaFalda				:= 53,
	Z_PosFuoriIngombroFalda 			:= 54,
	Z_PosStartLentaDepositoSuCatasta	:= 55,
	Z_PosDepositoInLentaSuCatasta		:= 56,
	Z_PosStartLentaDepositoFalda		:= 57,
	Z_PosDepositoInLentaFalda			:= 58,

	Z_PosStartLentaPrelievoLastra 		:= 101,
	Z_PosPrelievoInLentaLastra 			:= 102,
	Z_PosDistaccoLastraInLentaLastra	:= 103,
	Z_PosStartLentaDepositoLastra 		:= 104,
	Z_PosDepositoInLentaLastra			:= 105,
	Z_PosFuoriIngombroVuotoLastra		:= 106,
	
	Z_PosFuoriIngombroCaricoLastra		:= 126,
	Z_PosPostScarico					:= 127
);
END_TYPE

// ---- Data types/Programmi Movimento/GestioneEncoderEsterno.TcDUT
TYPE GestioneEncoderEsterno :
STRUCT
	Azzera : BOOL; //Comando di azzeramento encoder
	Pronto : BOOL; //Stato di encoder Pronto
	Direzione : bool; //Direzione di conteggio
END_STRUCT
END_TYPE

// ---- Data types/Programmi Movimento/MissionStateCase.TcDUT
TYPE MissionStateCase :
STRUCT
	Mission : e_Stato_Missione;		// Stato della missione
	NCase	: INT;		// Case dello stato della missione
	InitCase : BOOL;	// TRUE = case della missione inizializzato; FALSE= case della missione da inizializzare
END_STRUCT
END_TYPE

// ---- Data types/Programmi Movimento/Module_Palletizer_Aspirazione_IN.TcDUT
TYPE Module_Palletizer_Aspirazione_IN :
STRUCT
	PX_SuctionCupsUp : BOOL;
END_STRUCT
END_TYPE

// ---- Data types/Programmi Movimento/Module_Palletizer_Aspirazione_ManCmd.TcDUT
TYPE Module_Palletizer_Aspirazione_ManCmd :
STRUCT
	AttivazioneVuoto 	: BOOL;
	DisattivazioneVuoto : BOOL;
	SalitaVentose		: BOOL;
	DiscesaVentose		: BOOL;
	Home				: BOOL;
END_STRUCT
END_TYPE

// ---- Data types/Programmi Movimento/Module_Palletizer_AX_OUT.TcDUT
TYPE Module_Palletizer_AX_OUT :
STRUCT
	;
END_STRUCT
END_TYPE

// ---- Data types/Programmi Movimento/Module_Palletizer_AX_IN.TcDUT
TYPE Module_Palletizer_AX_IN :
STRUCT
	BeltSafety : BOOL;
	Px_Touch_1   : BOOL;
	Px_NuTouch	:BOOL ;
	Px_TouchEmergency_1	: BOOL;
	Px_Touch_2   : BOOL;
	Px_TouchEmergency_2	: BOOL;
	PX_GripPresence     : BOOL;
	Enable_TouchEmergency : POINTER TO BOOL;
	SimulazioneSenzaHW : bool;
END_STRUCT
END_TYPE

// ---- Data types/Programmi Movimento/Ax_Program_Parameters.TcDUT
TYPE Ax_Program_Parameters :
STRUCT
	Vel_Vuoto 			: REAL := 50; 		// Velocita di percorrenza tratto
	Acc_Vuoto 			: REAL := 50; 		// Accelerazione di percorrenza tratto
	Dec_Vuoto 			: REAL := 50; 		// Accelerazione di percorrenza tratto
	Jerk_Vuoto			: REAL := 100; 		// Jerk di percorrenza tratto
	Vel_Carico 			: REAL := 50; 		// Velocita di percorrenza tratto
	Acc_Carico 			: REAL := 50; 		// Accelerazione di percorrenza tratto
	Dec_Carico 			: REAL := 50; 		// Accelerazione di percorrenza tratto
	Jerk_Carico			: REAL := 100; 		// Jerk di percorrenza tratto
	Vel_Ridotta			: REAL := 5;		// Velocità ridotta per le fasi di approccio
	Torque				: REAL := 100;		// Coppia 
END_STRUCT
END_TYPE

// ---- Data types/Programmi Movimento/Descrittore_Programma.TcDUT
TYPE Descrittore_Programma :
STRUCT
	ID					: UINT := 9999; 	// Equivalente al n° di programma per riuscirlo a identificare
	Stato 				: UINT := 0; 		// 0=Non eseguito 1= Da Eseguire 2=In Esecuzione 3=Terminato 4=Interrotto 5=Annullato 6=Trasferito
	Quota_Destinazione 	: LREAL := 0; 		// Valore della posizione da raggiungere
	Velocita 			: REAL := 0; 		// Velocita di percorrenza tratto
	Accelerazione 		: REAL := 0; 		// Accelerazione di percorrenza tratto
	Decelerazione 		: REAL := 0; 		// Accelerazione di percorrenza tratto
	Jerk				: REAL := 0; 		// Jerk di percorrenza tratto
	Torque				: REAL := 0; 		// Coppia 
	DisabilitaTasteggio : BOOL := TRUE; 	// Controllo dei tastatori : TRUE= Tastatori abilitati, si genera errore in caso di tasteggio; FALSE = non si genera l'errore(utilizzato per i cicli falda e pallett)
	ControlloCoppiaAbilitato : BOOL := FALSE; //Modalita di funzionamento con controllo di coppia
	InnestoDiretto  : BOOL := FALSE; 		// Se TRUE, il programma corrente sovrascrive il programma in esecuzione
	InterpolaAsse	: INT := 0;				// 0: Nessuna Interpolazione,1: Interpolazione Asse,2: Interpolazione asse virtuale*)
END_STRUCT
END_TYPE

// ---- Data types/Programmi Movimento/Ax_Palletizer_Parameters.TcDUT
TYPE Ax_Palletizer_Parameters :
STRUCT
	HomeDefine		: REAL	:= 0.0;	(* Home Define (Posizione di Azzeramento Encoder) *)
	HomePosition	: REAL	:= 0.0;	(* Home Position (Posizione di Home) *)
	Vel				: REAL	:= 0.0;	(* Velocità di funzionamento*)
	Acc				: REAL	:= 100.0;	(* Accelerazione di funzionamento *)
	Dec				: REAL	:= 100.0;	(* Decelerazione di funzionamento *)
	Jerk			: REAL  := 100.0; (* Jerk di funzionamento *) 
	MaxTorque		: REAL	:= 100.0; (* Coppia massima utilizzata se si effettua il controllo di coppia*)
	JOGAcc			: REAL	:= 100.0;	(* Accelerazione di funzionamento *)
	JOGDec 			: REAL	:= 100.0;	(* Decelerazione di funzionamento *)
	MaxDeceleration : REAL  := 100.0; (* Massima Decelerazione *)
	MinPosition		: REAL	:= 0.0;
	MaxPosition		: REAL	:= 0.0;
	MaxVel		    : REAL  := 0.0; (* Massima velocità per gestire i jog manuali *)
	MaxAcc		    : REAL  := 0.0; (* Massima velocità per gestire i jog manuali *)
	MaxDec		    : REAL  := 0.0; (* Massima velocità per gestire i jog manuali *)
	ManSlowVel		: REAL	:= 0.0; (* Manual Slow Velocity (% of MaxVelocity) *)
	ManFastVel		: REAL	:= 0.0; (* Manual Fast Velocity (% of MaxVelocity) *)
	Quota_Destinazione	: LREAL  := 0.0; (*Posizione target da raggiungere*)
	HomeVelocity		: REAL  := 1.0; (* Velocità per ricerca sesore di Home *)
END_STRUCT
END_TYPE

// ---- Data types/Programmi Movimento/Module_Palletizer_Aspirazione_OUT.TcDUT
TYPE Module_Palletizer_Aspirazione_OUT :
STRUCT
	EV_Suction			: BOOL;
	EV_SuctionCupsUp	: BOOL;
	EV_SuctionCupsDown	: BOOL;
END_STRUCT
END_TYPE

// ---- Data types/Programmi Movimento/OffsetSicurezzaIngombro.TcDUT
TYPE OffsetSicurezzaIngombro :
STRUCT
	X: Offset_Sicurezza;
	Y: Offset_Sicurezza;
	Z: Offset_Sicurezza;
	J: Offset_Sicurezza;
END_STRUCT
END_TYPE

// ---- Data types/Programmi Movimento/OffsetDistacco.TcDUT
TYPE OffsetDistacco :
STRUCT
	Lastra 	: StrutturaGenericaQuotaAssi; 
	Falda 	: StrutturaGenericaQuotaAssi;
END_STRUCT
END_TYPE

// ---- Data types/Programmi Movimento/Offset_Pass_Mode.TcDUT
TYPE Offset_Pass_Mode :
STRUCT
	X	: REAL := 100; // mm di pass mode
	Y	: REAL := 0; // mm di pass mode
	Z	: REAL := 100; // mm di pass mode
	J	: REAL := 0; // ° di pass mode
END_STRUCT
END_TYPE

// ---- Data types/Programmi Movimento/Offset_Prelievi_Lenti.TcDUT
TYPE Offset_Prelievi_Lenti :
STRUCT
	Pallet						: REAL := 200;	// Offset utilizzato in fase di prelievo pallet per dare inizio alla discesa lenta
	Falde						: REAL := 100;	// Offset utilizzato in fase di prelievo falda per dare inizio alla discesa lenta 
	Pacco						: REAL := 200;  // Offset utilizzato in fase di prelievo pacco per dare inizio alla discesa lenta 
END_STRUCT
END_TYPE

// ---- Data types/Programmi Movimento/Offeset_Apprendimento.TcDUT
TYPE Offeset_Apprendimento :
STRUCT
	Lastra 	: StrutturaGenericaQuotaAssi;
	Falda 	: StrutturaGenericaQuotaAssi;
END_STRUCT
END_TYPE

// ---- Data types/Programmi Movimento/Offset_Sicurezza.TcDUT
TYPE Offset_Sicurezza :
STRUCT
	Carico		: REAL := 100;  // OFFSET di sicurezza utilizzato per il calcolo della quota di fuoringombro dell'asse 
	Avuoto		: REAL := 100;  // OFFSET di sicurezza utilizzato per il calcolo della quota di fuoringombro dell'asse 

END_STRUCT
END_TYPE

// ---- Data types/Programmi Movimento/Offset_Sicurezza_Anticipo_Movimenti.TcDUT
TYPE Offset_Sicurezza_Anticipo_Movimenti :
STRUCT
	OffsetSicurezzaAnticipo_X : REAL := 100; 
	OffsetSicurezzaAnticipo_Y : REAL := 100; 
	OffsetSicurezzaAnticipo_Z : REAl := 100;
END_STRUCT
END_TYPE

// ---- Data types/Programmi Movimento/Overide_Dinamico.TcDUT
TYPE Overide_Dinamico :
STRUCT
	NTrasportiOccupati : ARRAY[1..MAXSOGLIEOVERRIDE] OF UINT;	// N° Trasporti occupati paertendo dal ribaltino che stabilisce la soglia i-esima di velocità
	Override : ARRAY[1..MAXSOGLIEOVERRIDE] OF REAL; //Ovverride Relativo alla soglia i-esima
END_STRUCT
END_TYPE

// ---- Data types/Programmi Movimento/ProgrammaLog.TcDUT
TYPE ProgrammaLog :
STRUCT
	Programma : ARRAY[0..10] OF Descrittore_Programma;
END_STRUCT
END_TYPE

// ---- Data types/Programmi Movimento/Stato_Ciclo_Lavoro.TcDUT
TYPE Stato_Ciclo_Lavoro :
STRUCT
	Stato : UINT := 0; // 0=Non eseguito 1=In Esecuzione 2=Terminato
	Passo : UINT := 0;
	PassoDopoInterruzzione	: UINT := 0;
END_STRUCT
END_TYPE

// ---- Data types/Programmi Movimento/StrutturaGenericaQuotaAssi.TcDUT
TYPE StrutturaGenericaQuotaAssi :
STRUCT
	X : LREAL := 20;
	Y : LREAL := 20;
	Z : LREAL := 20;
	J : LREAL := 2;

END_STRUCT
END_TYPE

// ---- Data types/Programmi Movimento/TFDimensioniPinza.TcDUT
TYPE TFDimensioniPinza :
STRUCT
	Lunghezza : REAL := 1600; // Lunghezza Corpo pinza - Dimensione lungo X (da centro trave)
	Larghezza : REAL := 1600; // Larghezza Corpo pinza - Dimensione Lungo Y (da centro trave)
	Spessore  : REAL := 200; // Spessore Corpo Pinza - Dimensione Lungo Z (da centro di rotazione)
	DimTraveVerticale : REAL := 150; //Dimensione Trave Verticale
END_STRUCT
END_TYPE

// ---- Data types/Programmi Movimento/TFMachinePalletizer_ModuleState.TcDUT
TYPE TFMachinePalletizer_ModuleState :
STRUCT
	Cmd	  : UDINT;
	CmdCase : UDINT;
	Error : UDINT;
	ErrorExtra : UDINT;
END_STRUCT
END_TYPE

// ---- Data types/Programmi Movimento/TFMachinePalletizer_MachineState.TcDUT
TYPE TFMachinePalletizer_MachineState :
STRUCT
	Cmd	  : UDINT;
	CmdCase : UDINT;
	Error : UDINT;
	ErrorExtra : UDINT;

	Auto : BOOL;
	Run : BOOL;
	EmergencyOK : BOOL;
	PowerOK	: BOOL;
	
END_STRUCT
END_TYPE

// ---- Data types/Programmi Movimento/TFMachinePalletizer_VelocityOverride_TF.TcDUT
TYPE TFMachinePalletizer_VelocityOverride_TF :
STRUCT
	
	Auto		: REAL	:= 50.0;	(* READ	- (%) In Auto, è l'override degli override, con questo si abbassa la velocità globale di tutti i cicli *)
	Jog			: REAL	:= 10.0;	(* READ	- (%) In Jog *)
	Pack		: REAL	:= 50.0;	(* READ	- (%) Relativo al ciclo pacco *)
	Pallet		: REAL	:= 50.0;	(* READ	- (%) Relativo al ciclo pallet *)
	Layer		: REAL	:= 50.0;	(* READ	- (%) Relativo al ciclo falda *)
	Riposo		: REAL  := 50.0;	(* READ	- (%) Relativo al ciclo di riposo *)
	
END_STRUCT
END_TYPE

// ---- Data types/Programmi Movimento/TFModulePalletizerRobot_Point_TF.TcDUT
TYPE TFModulePalletizerRobot_Point_TF :
STRUCT
	
	X				: LREAL	:= 0.0;	(* X Position *)
	Y				: LREAL	:= 0.0;	(* Y Position *)
	Z				: LREAL	:= 0.0;	(* Z Position *)
	J				: LREAL	:= 0.0;	(* J Position *)
	K				: LREAL	:= 0.0;	(* K Position *)
	
END_STRUCT
END_TYPE

// ---- Data types/Programmi Movimento/TFModulePalletizerSTATUS_TF.TcDUT
TYPE TFModulePalletizerSTATUS_TF :
STRUCT
	
	X	: TFMachinePalletizer_AxeState_TF;	(* X Axe State (UI Position=mm, UI Velocity=mm/sec UI Acc/Dec=mm/sec2) *)
	Y	: TFMachinePalletizer_AxeState_TF;	(* Y Axe State (UI Position=mm, UI Velocity=mm/sec UI Acc/Dec=mm/sec2) *)
	Z	: TFMachinePalletizer_AxeState_TF;	(* Z Axe State (UI Position=mm, UI Velocity=mm/sec UI Acc/Dec=mm/sec2) *)
	J	: TFMachinePalletizer_AxeState_TF;	(* J Axe State (UI Position=°,  UI Velocity=°/sec  UI Acc/Dec=°/sec2) *)
	K	: TFMachinePalletizer_AxeState_TF;	(* K Axe State (UI Position=mm, UI Velocity=mm/sec UI Acc/Dec=mm/sec2) *)
	
	ModAsse_X : TFMachinePalletizer_ModuleState;
	ModAsse_Y : TFMachinePalletizer_ModuleState;
	ModAsse_Z : TFMachinePalletizer_ModuleState;
	ModAsse_J : TFMachinePalletizer_ModuleState;
	ModAsse_K : TFMachinePalletizer_ModuleState;
	
	Macchina : TFMachinePalletizer_MachineState;
	
	ModAspirazione : TFMachinePalletizer_ModuleState;
	
	Pinza : TFMAchinePalletizer_PinzaVentoseStatus;

END_STRUCT
END_TYPE

// ---- Data types/Programmi Movimento/TFTraiettoria.TcDUT
TYPE TFTraiettoria :
STRUCT
	PuntoDiApproccioStartPoint 			: TFModulePalletizerRobot_Point_TF;			// Punto Precedente al punto iniziale, utilizzato per la lenta in fase di prelievo falda e pallet lastra
	StartPoint 							: TFModulePalletizerRobot_Point_TF;			// Punto iniziale
	PuntoDiPostPosizionamentoStartPoint : TFModulePalletizerRobot_Point_TF;			// Punto Successivo al punto iniziale, utilizzato per la lenta in fase di distacco dopo il prelievo elemento

	PuntoIntermedio 	: ARRAY[1..MAXTPOINTS] OF TFModulePalletizerRobot_Point_TF;	// Punti Intermedi
	PassModePoint_X		: ARRAY[1..MAXTPOINTS] OF REAL;								// Quota di anticipo asse X per innescare movimento successivo	
	PassModePoint_Y		: ARRAY[1..MAXTPOINTS] OF REAL;								// Quota di anticipo asse Y per innescare movimento successivo	
	PassModePoint_Z		: ARRAY[1..MAXTPOINTS] OF REAL;								// Quota di anticipo asse Z per innescare movimento successivo	
	PassModePoint_J		: ARRAY[1..MAXTPOINTS] OF REAL;								// Quota di anticipo asse J per innescare movimento successivo	
	PassModePoint_K		: ARRAY[1..MAXTPOINTS] OF REAL;								// Quota di anticipo asse K per innescare movimento successivo	
	PassModePoint_X_Enable	 : ARRAY[1..MAXTPOINTS] OF BOOL;				// Abilitazione del singolo pass mode(relativo al punto i-esimo)
	PassModePoint_Y_Enable	 : ARRAY[1..MAXTPOINTS] OF BOOL;				// Abilitazione del singolo pass mode(relativo al punto i-esimo)
	PassModePoint_Z_Enable	 : ARRAY[1..MAXTPOINTS] OF BOOL;				// Abilitazione del singolo pass mode(relativo al punto i-esimo)
	PassModePoint_J_Enable	 : ARRAY[1..MAXTPOINTS] OF BOOL;				// Abilitazione del singolo pass mode(relativo al punto i-esimo)
	PassModePoint_K_Enable	 : ARRAY[1..MAXTPOINTS] OF BOOL;				// Abilitazione del singolo pass mode(relativo al punto i-esimo)
	PuntoDiApproccioEndPoint : TFModulePalletizerRobot_Point_TF;			// Punto di approccio in fase di deposito
	EndPoint				 : TFModulePalletizerRobot_Point_TF;			// Punto finale
	
	PuntoDiApproccioSecondarioEndPoint	: TFModulePalletizerRobot_Point_TF;			// Punto di approccio in fase di deposito SECONDARIO, SE è PREVISTO IL DEPOSITO FALDA
	EndPointSecondario					: TFModulePalletizerRobot_Point_TF;			// Punto finale deposito SECONDARIO, SE è PREVISTO IL DEPOSITO LASTRA
	
	PassModeGlobalEnable 	 : BOOL;										// Abilitazione globale del pass mode
END_STRUCT
END_TYPE

// ---- Data types/Programmi Movimento/TFWorkAreaManager.TcDUT
TYPE TFWorkAreaManager :
STRUCT
	State : e_Stato_WAManager := -1;	//Stato
END_STRUCT
END_TYPE

// ---- Data types/Programmi Movimento/Work_PickPoint_Dimension.TcDUT
TYPE Work_PickPoint_Dimension :
STRUCT
	Xdim	:REAL := 600; // Larghezza
	Ydim	:REAL := 0; // Lunghezza
	Zdim	:REAL := 900; // Altezza
END_STRUCT
END_TYPE

// ---- Data types/Scambio Dati Trasporti/DUT_ArrayPacchi.TcDUT
TYPE DUT_ArrayPacchi :
STRUCT
	Pacco :ARRAY[1..MAXDIMARRAYPACCHI] OF DUT_Struttura_Dati_Pacco;
END_STRUCT
END_TYPE

// ---- Data types/Scambio Dati Trasporti/DUT_Lista_Pacchi_In_Pila.TcDUT
TYPE DUT_Lista_Pacchi_In_Pila :
STRUCT
	ID_Pacco : ARRAY[0..MAXHANDLINGSTACK-1] OF UDINT;
END_STRUCT
END_TYPE

// ---- Data types/Scambio Dati Trasporti/DUT_Struttura_Dati_Pacco.TcDUT
TYPE DUT_Struttura_Dati_Pacco :
STRUCT

	ID			: DUT_Lista_Pacchi_In_Pila;
	PC			: UINT;					(* Production Code *)
	PP      	: BOOL; 				(* Pack Presence *)

	X 			: REAL;					(* X dimension *)
	Y 			: REAL;					(* Y dimension *)
	Z 			: REAL;					(* Z dimension *)
	
END_STRUCT
END_TYPE

// ---- Data types/StatoLineaDepal.TcDUT
TYPE StatoLineaDepal :
STRUCT
	AsseX	: TFMachinePalletizer_AxeState_TF;	(* X Axe State (UI Position=mm, UI Velocity=mm/sec UI Acc/Dec=mm/sec2) *)
	AsseY	: TFMachinePalletizer_AxeState_TF;	(* Y Axe State (UI Position=mm, UI Velocity=mm/sec UI Acc/Dec=mm/sec2) *)
	AsseZ	: TFMachinePalletizer_AxeState_TF;	(* Z Axe State (UI Position=mm, UI Velocity=mm/sec UI Acc/Dec=mm/sec2) *)
	AsseJ	: TFMachinePalletizer_AxeState_TF;	(* J Axe State (UI Position=°,  UI Velocity=°/sec  UI Acc/Dec=°/sec2) *)

	DepalAuto 		: BOOL;	//Indica che il Depal è in automatico
	DepalError 		: UDINT;	//Se <> 0 identifica il codice di errore della macchina

	RulliereInterneAuto 	: BOOL; //Indica che le rulliere interne sono in automatico
	RulliereInterneError 	: UDINT; //Se <> 0 identifica il codice di errore della macchina

	RulliereEsterneAuto 	: BOOL; //Indica che le rulliere esterne sono in automatico
	RulliereEsterneError 	: UDINT; //Se <> 0 identifica il codice di errore della macchina
	
	ElementoSuRullieraPrelievo1 : TFMachineTransportElement;
	ElementoSuRullieraPrelievo2 : TFMachineTransportElement;
	testnum : REAL;
		
END_STRUCT
END_TYPE

// ---- Data types/Strutture Aggiornate/TFMachinePalletizer_FormingForSlab.TcDUT
TYPE TFMachinePalletizer_FormingForSlab :
STRUCT
	Enable		: INT							:= -1;	(* Formatura Abilitata 0=no, 1=si, -1 dato non valido *)
	Code		: ARRAY[1..MAXFORMINGCODE] 		OF INT;	(* Codici di Pallettizzazione (0..n=, -1 dato non valido) *)
	Pallet		: TFMachinePalletizer_Pallet;	(* Pallet assegnato (0 = tipo 0, 1 = tipo 1, 2 = tipo 2,  …. , 0 / -1 dato non valido *)
	LGVAttr		: INT							:= -1;  (* Attributi LGV (-1= non valido) *)
	PElement	: ARRAY[1..MAXFORMINGSLAB] OF TFMachinePalletizer_PlaceElement; (* Elemento i-esimo da dapositare *)
	
	AuxAttr		: INT 							:= -1;	(* Attributi Ausiliari per la gestione di abilitazioni varie 
															-> Bit 0 : Abilitazione BARCODE 
															-> Bit 1 : ABilita PRESA FALDA CON ARPIONI*)
															
	GUID		: UINT							:= 0;	(* Identificatore univoco della Formatura *)
END_STRUCT
END_TYPE

// ---- Data types/Strutture Aggiornate/TFMachinePalletizer_Layer.TcDUT
TYPE TFMachinePalletizer_Layer :
STRUCT
	Tipologia	: INT	:= -1;  (* Indica la tipologia dell'elemento *)
	Code		: INT   := -1;  (* Indica il codice della falda *)
	TPick		: INT	:= -1;	(* Tipologia di presa della falda,*)
	XDim		: REAL	:= 0.0;	(* (mm) Dimensione X *)
	YDim		: REAL	:= 0.0;	(* (mm) Dimensione Y *)
	ZDim		: REAL	:= 0.0;	(* (mm) Dimensione Z *)
	
	//OffsetDep_0 	: TFMachinePalletizer_OffsetElement; (* OFFSET di deposito, utilizzato per lato 0-90 *)
	//OffsetDep_90 	: TFMachinePalletizer_OffsetElement; (* OFFSET di deposito, utilizzato per CASSE *)
	//OffsetDep_180 	: TFMachinePalletizer_OffsetElement; (* OFFSET di deposito, utilizzato per lato 90-180 *)
	
END_STRUCT
END_TYPE

// ---- Data types/Strutture Aggiornate/TFMachinePalletizer_Mission.TcDUT
TYPE TFMachinePalletizer_Mission :
STRUCT
	
	State			: e_Stato_Missione	:= MISSION_STATE_NOP; (* Stato Missione *)
	PPick			: UINT	:= 0;		(* Puntatore Tabella WorkPickPoint(Lastra)/WorkArea(Lastra/LAYER) *)
	TPick			: e_Tipo_PresaEndEffector	:= 0;		(* Tipo di Prelievo: 0=Pick From PickPoint (PACCO), 1=Pick From WorkArea (PALLET), 2=Pick From WorkArea (FALDA) *)
	PPlace			: UINT	:= 0;		(* Puntatore Tabella WorkArea *)
	
	XPick			: LREAL	:= 0.0;		(* (mm) Punto di Prelievo X - Quota assoluta di impianto DA ORIGINE *)
	YPick			: LREAL	:= 0.0;		(* (mm) Punto di Prelievo Y - Quota assoluta di impianto DA ORIGINE *)
	ZPick			: LREAL	:= 0.0;		(* (mm) Punto di Prelievo Z - Quota assoluta di impianto DA ORIGINE *)
	JPick			: LREAL	:= 0.0;		(* (mm) Punto di Prelievo - Quota di Rotazione lungo asse X *)
	KPick			: LREAL	:= 0.0;		(* (mm) Punto di Prelievo - Quota di Rotazione lungo asse Y *)
	WPick			: LREAL	:= 0.0;		(* (mm) Punto di Prelievo - Quota di Rotazione lungo asse Z *)

	XPickApproach	: LREAL	:= 0.0;		(* (mm) Punto di Approccio X - Quota assoluta di impianto DA ORIGINE *)
	YPickApproach	: LREAL	:= 0.0;		(* (mm) Punto di Approccio Y - Quota assoluta di impianto DA ORIGINE *)
	ZPickApproach	: LREAL	:= 0.0;		(* (mm) Punto di Approccio Z - Quota assoluta di impianto DA ORIGINE *)
	JPickApproach	: LREAL	:= 0.0;		(* (mm) Punto di Approccio - Quota di Rotazione lungo asse X *)
	KPickApproach	: LREAL	:= 0.0;		(* (mm) Punto di Approccio - Quota di Rotazione lungo asse Y *)
	WPickApproach	: LREAL	:= 0.0;		(* (mm) Punto di Approccio - Quota di Rotazione lungo asse Z *)
	
	XPlace			: LREAL	:= 0.0;		(* (mm) Punto di Deposito X - Quota assoluta di impianto DA ORIGINE *)
	YPlace			: LREAL	:= 0.0;		(* (mm) Punto di Deposito Y - Quota assoluta di impianto DA ORIGINE *)
	ZPlace			: LREAL	:= 0.0;		(* (mm) Punto di Deposito Z - Quota assoluta di impianto DA ORIGINE *)
	JPlace			: LREAL	:= 0.0;		(* (mm) Punto di Deposito - Quota di Rotazione lungo asse X *)
	KPlace			: LREAL	:= 0.0;		(* (mm) Punto di Deposito - Quota di Rotazione lungo asse Y *)
	WPlace			: LREAL	:= 0.0;		(* (mm) Punto di Deposito - Quota di Rotazione lungo asse Z *)

	XPlaceApproach	: LREAL	:= 0.0;		(* (mm) Punto di Approccio X - Quota assoluta di impianto DA ORIGINE *)
	YPlaceApproach	: LREAL	:= 0.0;		(* (mm) Punto di Approccio Y - Quota assoluta di impianto DA ORIGINE *)
	ZPlaceApproach	: LREAL	:= 0.0;		(* (mm) Punto di Approccio Z - Quota assoluta di impianto DA ORIGINE *)
	JPlaceApproach	: LREAL	:= 0.0;		(* (mm) Punto di Approccio - Quota di Rotazione lungo asse X *)
	KPlaceApproach	: LREAL	:= 0.0;		(* (mm) Punto di Approccio - Quota di Rotazione lungo asse Y *)
	WPlaceApproach	: LREAL	:= 0.0;		(* (mm) Punto di Approccio - Quota di Rotazione lungo asse Z *)
	
	(* Deposito secondario utilizzato per depositi intermedi -> Es. x falda *)
	XPlaceSecondario			: LREAL	:= 0.0;		(* (mm) Punto di Deposito X Secondario - Quota assoluta di impianto DA ORIGINE *)
	YPlaceSecondario			: LREAL	:= 0.0;		(* (mm) Punto di Deposito Y Secondario - Quota assoluta di impianto DA ORIGINE *)
	ZPlaceSecondario			: LREAL	:= 0.0;		(* (mm) Punto di Deposito Z Secondario - Quota assoluta di impianto DA ORIGINE *)
	JPlaceSecondario			: LREAL	:= 0.0;		(* (mm) Punto di Deposito Secondario - Quota di Rotazione lungo asse X *)
	KPlaceSecondario			: LREAL	:= 0.0;		(* (mm) Punto di Deposito Secondario - Quota di Rotazione lungo asse Y *)
	WPlaceSecondario			: LREAL	:= 0.0;		(* (mm) Punto di Deposito Secondario - Quota di Rotazione lungo asse Z *)

	XPlaceApproachSecondario	: LREAL	:= 0.0;		(* (mm) Punto di Approccio X Secondario- Quota assoluta di impianto DA ORIGINE *)
	YPlaceApproachSecondario	: LREAL	:= 0.0;		(* (mm) Punto di Approccio Y Secondario- Quota assoluta di impianto DA ORIGINE *)
	ZPlaceApproachSecondario	: LREAL	:= 0.0;		(* (mm) Punto di Approccio Z Secondario- Quota assoluta di impianto DA ORIGINE *)
	JPlaceApproachSecondario	: LREAL	:= 0.0;		(* (mm) Punto di Approccio Secondario- Quota di Rotazione lungo asse X *)
	KPlaceApproachSecondario	: LREAL	:= 0.0;		(* (mm) Punto di Approccio Secondario- Quota di Rotazione lungo asse Y *)
	WPlaceApproachSecondario	: LREAL	:= 0.0;		(* (mm) Punto di Approccio Secondario- Quota di Rotazione lungo asse Z *)

	XDim			: REAL	:= 0.0;		(* (mm) Dimensione X del Lastra/Pallet/Falda *)
	YDim			: REAL	:= 0.0;		(* (mm) Dimensione Y del Lastra/Pallet/Falda *)
	ZDim			: REAL	:= 0.0;		(* (mm) Dimensione Z del Lastra/Pallet/Falda *)
	
	Slab			: TFMachinePalletizer_PlaceElement; (* Struttura Usata per Tracciare l'elemento presente in pinza *)

END_STRUCT
END_TYPE

// ---- Data types/Strutture Aggiornate/TFMachinePalletizer_Pallet.TcDUT
TYPE TFMachinePalletizer_Pallet :
STRUCT
	Tipologia				: INT	:= 0;  (* Indica la tipologia dell'elemento *)
	Code					: INT 	:= -1;	(* Codici Del supporto *)
	XDim					: REAL	:= 0.0;	(* (mm) Dimensione X ex Lunghezza_Cavallina*) // Lunghezza X della cavallina (Lunghezza per la cassa)
	YDim					: REAL	:= 0.0;	(* (mm) Dimensione Y ex L_Base *) // Larghezza totale della base della cavallina (Larghezza della cassa)
	ZDim					: REAL	:= 0.0;	(* (mm) Dimensione Z Base Cavallina(interno, + bassa) o Base Cassa *)
	ZDim_Ext1 				: REAL  := 0.0; (* (mm) Dimensione Z Base Cavallina(esterna, + alta) NON USATA PER CASSA *)
	HMAX					: REAL  := 0.0;	(* (mm) Altezza Massima dell'elemento telaio cavallina o sponde cassa, dal terreno alla massima altezza*)
	
	//ZDim_Int1 				: REAL  := 0.0; // Altezza della base interna 1 della cavallina (altezza della base di supporto per la cassa) 
	//ZDim_Int2 				: REAL  := 0.0; // Altezza della base interna 2 della cavallina
	//ZDim_Ext2 				: REAL  := 0.0; // Altezza della base esterna 2 della cavallina
	
	DimVertice 					: REAL  := 0.0; // Larghezza parte alta della cavallina
	DimBaseUtile 				: REAL  := 0.0; // Larghezza della base utile di appoggio delle lastre x cavallina
	TipoTrabajoLado_Cavallete 	: INT := 0; // // 0-trabaja aambos lados 1-Lado 0 Grados 2-Lado 180 Grados
	
	AltezzaDenteRitenuta		: REAL := 0.0; 	(* (mm) Altezza del dente di ritenuta (per cavalletti) *)
	TipoPianoAppoggio			: UINT := 0; //0=Con dente di ritenuta e in piano, 1=piano inclinato
	//Spessore_DenteRitenuta	: REAL := 0.0;	(* (mm) Spessore del dente di ritenuta (per cavalletti) *)
	//OffsetY_DenteRitenuta 	: REAL := 0.0;	(* (mm) Posizione del dente di ritenuta rispetto la quota Y del cavalletto (per cavalletti) *)
	
	LatoDeposito 			: UINT := 0; 	(* Lato in cui depositare gli elementi in caso di tipologia BUNDLE 0 o 180 *)
	AngoloAlfaBundle		: REAL := 0.0;	(* Angolo Alfa di inclinazione del BUNDLE *)
	
	OFSDE_X90 				: REAL := 0.0;	(* (mm) OFFSET di deposito direzione X, utilizzato per PALLET o CASSE *)
	OFSDE_Y90 				: REAL := 0.0;	(* (mm) OFFSET di deposito direzione Y, utilizzato per PALLET o CASSE *)
	OFSDE_Z90 				: REAL := 0.0;	(* (mm) OFFSET di deposito direzione Z, utilizzato per PALLET o CASSE *)
	OFSDE_J90 				: REAL := 0.0;	(* (mm) OFFSET di deposito direzione J, utilizzato per PALLET o CASSE *)
	
	OFSDE_X0 				: REAL := 0.0;	(* (mm) OFFSET di deposito direzione X, utilizzato per CAVALLETTI *)
	OFSDE_Y0 				: REAL := 0.0;	(* (mm) OFFSET di deposito direzione Y, utilizzato per CAVALLETTI *)
	OFSDE_Z0 				: REAL := 0.0;	(* (mm) OFFSET di deposito direzione Z, utilizzato per CAVALLETTI *)
	OFSDE_J0 				: REAL := 0.0;	(* (mm) OFFSET di deposito direzione J, utilizzato per CAVALLETTI *)
	
	OFSDE_X180 				: REAL := 0.0;	(* (mm) OFFSET di deposito direzione X, utilizzato per CAVALLETTI *)
	OFSDE_Y180 				: REAL := 0.0;	(* (mm) OFFSET di deposito direzione Y, utilizzato per CAVALLETTI *)
	OFSDE_Z180 				: REAL := 0.0;	(* (mm) OFFSET di deposito direzione Z, utilizzato per CAVALLETTI *)
	OFSDE_J180 				: REAL := 0.0;	(* (mm) OFFSET di deposito direzione J, utilizzato per CAVALLETTI *)

	ConfigurazioneBC 	 	: INT := -1;	(* (mm) Indica la modalità di funzionamento del barcode.. sono i suoi parametri *)
	QuotaRilevamentoBC_X 	: REAL := 0;	(* (mm) Indica la posizione del barcode lungo la sua lunghezza e rispetto il punto medio *)
	QuotaRilevamentoBC_Y 	: REAL := 0;	(* (mm) Indica la posizione del barcode lungo la sua larghezza e rispetto il punto medio	*)
	QuotaRilevamentoBC_Z 	: REAL := 0;	(* (mm) Indica la posizione del barcode lungo il suo spessore e rispetto il punto medio *)
	QuotaRilevamentoBC_J 	: REAL := 0;	(* (mm) Indica la posizione del barcode lungo il suo spessore e rispetto il punto medio *)
END_STRUCT
END_TYPE

// ---- Data types/Strutture Aggiornate/TFMachinePalletizer_PalletSlabOld.TcDUT
TYPE TFMachinePalletizer_PalletSlabOld :
STRUCT
	Tipologia	: INT	:= 0;  (* Indica la tipologia dell'elemento *)
	Code		: INT 	:= -1;	(* Codici Della *)
	XDim		: REAL	:= 0.0;	(* (mm) Dimensione X *)
	YDim		: REAL	:= 0.0;	(* (mm) Dimensione Y *)
	ZDim		: REAL	:= 0.0;	(* (mm) Dimensione Z Base Cavallina o Base Cassa *)
	HMAX		: REAL  := 0.0;	(* (mm) Altezza Massima dell'elemento telaio cavallina o sponde cassa *)
	
	AltezzaDenteRitenuta	: REAL := 0.0; 	(* (mm) Altezza del dente di ritenuta (per cavalletti) *)
	Spessore_DenteRitenuta	: REAL := 0.0;	(* (mm) Spessore del dente di ritenuta (per cavalletti) *)
	OffsetY_DenteRitenuta 	: REAL := 0.0;	(* (mm) Posizione del dente di ritenuta rispetto la quota Y del cavalletto (per cavalletti) *)

	DimBaseUtile			: REAL := 0.0;
	DimVertice				: REAL := 0.0;
	TipoPianoAppoggio		: uint := 0; //0=Con dente di ritenuta e in piano, 1=piano inclinato

	
	OFSDE_X90 				: REAL := 0.0;	(* (mm) OFFSET di deposito direzione X, utilizzato per PALLET o CASSE *)
	OFSDE_Y90 				: REAL := 0.0;	(* (mm) OFFSET di deposito direzione Y, utilizzato per PALLET o CASSE *)
	OFSDE_Z90 				: REAL := 0.0;	(* (mm) OFFSET di deposito direzione Z, utilizzato per PALLET o CASSE *)
	OFSDE_J90 				: REAL := 0.0;	(* (mm) OFFSET di deposito direzione J, utilizzato per PALLET o CASSE *)
	
	OFSDE_X0 				: REAL := 0.0;	(* (mm) OFFSET di deposito direzione X, utilizzato per CAVALLETTI *)
	OFSDE_Y0 				: REAL := 0.0;	(* (mm) OFFSET di deposito direzione Y, utilizzato per CAVALLETTI *)
	OFSDE_Z0 				: REAL := 0.0;	(* (mm) OFFSET di deposito direzione Z, utilizzato per CAVALLETTI *)
	OFSDE_J0 				: REAL := 0.0;	(* (mm) OFFSET di deposito direzione J, utilizzato per CAVALLETTI *)
	
	OFSDE_X180 				: REAL := 0.0;	(* (mm) OFFSET di deposito direzione X, utilizzato per CAVALLETTI *)
	OFSDE_Y180 				: REAL := 0.0;	(* (mm) OFFSET di deposito direzione Y, utilizzato per CAVALLETTI *)
	OFSDE_Z180 				: REAL := 0.0;	(* (mm) OFFSET di deposito direzione Z, utilizzato per CAVALLETTI *)
	OFSDE_J180 				: REAL := 0.0;	(* (mm) OFFSET di deposito direzione J, utilizzato per CAVALLETTI *)

	ConfigurazioneBC 	 : INT := -1;	(* (mm) Indica la modalità di funzionamento del barcode.. sono i suoi parametri *)
	QuotaRilevamentoBC_X : REAL := 0;	(* (mm) Indica la posizione del barcode lungo la sua lunghezza e rispetto il punto medio *)
	QuotaRilevamentoBC_Y : REAL := 0;	(* (mm) Indica la posizione del barcode lungo la sua larghezza e rispetto il punto medio	*)
	QuotaRilevamentoBC_Z : REAL := 0;	(* (mm) Indica la posizione del barcode lungo il suo spessore e rispetto il punto medio *)
	QuotaRilevamentoBC_J : REAL := 0;	(* (mm) Indica la posizione del barcode lungo il suo spessore e rispetto il punto medio *)

END_STRUCT
END_TYPE

// ---- Data types/Strutture Aggiornate/TFMachinePalletizer_WorkAreaState_VECCHIO.TcDUT
TYPE TFMachinePalletizer_WorkAreaState_VECCHIO :
STRUCT
	State		: e_Stato_WorkArea	:= WORKAREA_STATE_FREE_DISABLED;	(* Stato Area di Lavoro/Piazzola
																			(0=Assente e Area Disabilitata,
																			1=Presente e Area Disabilitata,
																			2=Assente in Lavorazione,
																			3=Presente in Lavorazione,
																			4=Presente con Pallettizzazione Terminata,
																			5=Presente con Pallettizzazione Terminata e Area Disabilitata,
																			6=Presente in Nastratura,
																			7=Presente in Nastratura e Area Disabilitata,
																			8=Presente con Nastratura Terminata,
																			9=Presente con Nastratura Terminata e Area Disabilitata,
																			10=Presente con Lavorazione Terminata,
																			11=Presente con Lavorazione Terminata e Area Disabilitata,
																			12=Presente con LGV in Richiesta Ingresso,
																			13=Presente con LGV in Richiesta Ingresso e Area Disabilitata,
																			14=Presente con LGV in Ingombro,
																			15=Presente con LGV in Ingombro e Area Disabilitata,
																			16=Presente con LGV Fuori Ingombro e Pallet Estratto,
																			17=Presente con LGV Fuori Ingombro e Pallet Estratto e Area Disabilitata, NOT USED !!!!!!!!!!!
																			99=Errore
																			-1 dato non valido) *)
	F			: INT	:= -1;	(* Forming Pointer - Puntatore tabella formature (1..n=, -1 dato non valido *)
	P			: INT	:= -1;	(* Pack Pointer - Puntatore tabella LASTRE (0..n-1=, -1 dato non valido),Numero lastra successiva da depositare *)
	//L			: INT	:= -1;	(* Codice Layer da depositare in Layer Orrizontale o cavalletto lato 0°(0=Da Depositare, 1=Depositato o Nessun Layer Previsto, -1= dato non valido *)
	//NL			: INT	:= -1;	(* Numero Layer depositati in Orrizontale o su cavalletto lato 90° *)
	//L2			: INT 	:= -1;	(* Codice Layer da depositare su cavalletto lato 180° (0=Da Depositare, 1=Depositato o Nessun Layer Previsto, -1= dato non valido *)
	//NL2			: INT	:= -1;	(* Numero Layer depositati su cavalletto lato 180° *)
	//PN			: INT	:= -1;	(* Positive/Negative Pointer - Puntatore tabella pacchi Positiva/Negativa (0=Positiva, 1=Negativa, -1 dato non valido *)
	PackPointerModified	: BOOL	:= FALSE;		(* Se TRUE, indica che è stata effettuata una modfica sui dati della WA da parte dell' HMI (Settata da HMI e resettata da PLC) *)
	PackPointer			: INT	:= -1;			(* Rappresenta l'indice del pacco da depositare dopo modfica manuale,cioè con PackPointerModified=TRUE *)
	//NLP			: ARRAY[1..MAXFORMINGPACK] OF INT;//   := -1;	(* Numero di Falde depositate sul Pacco/Lastra *)
	Slab		: ARRAY[1..MAXFORMINGSLAB] OF TFMachinePalletizer_PlaceElement; (* Struttura Usata per Tracciare Gli Elementi Depositati sulla Workarea *)
	LGVAttr		: INT;
	BCRead		: ARRAY[1..MAXNUMBARCODE] OF TFMachinePalletizer_BarCode;

END_STRUCT
END_TYPE

// ---- Data types/Strutture Aggiornate/TFMachinePalletizer_WorkAreaState.TcDUT
TYPE TFMachinePalletizer_WorkAreaState :
STRUCT
	ID				: LINT; (* Identificatore univoco dell'oggetto sulla WorkArea *)
	State			: e_Stato_WorkArea	:= WORKAREA_STATE_FREE_DISABLED;	(* Stato Area di Lavoro/Piazzola
																			(0=Assente e Area Disabilitata,
																			1=Presente e Area Disabilitata,
																			2=Assente in Lavorazione,
																			3=Presente in Lavorazione,
																			4=Presente con Pallettizzazione Terminata,
																			5=Presente con Pallettizzazione Terminata e Area Disabilitata,
																			6=Presente in Nastratura,
																			7=Presente in Nastratura e Area Disabilitata,
																			8=Presente con Nastratura Terminata,
																			9=Presente con Nastratura Terminata e Area Disabilitata,
																			10=Presente con Lavorazione Terminata,
																			11=Presente con Lavorazione Terminata e Area Disabilitata,
																			12=Presente con LGV in Richiesta Ingresso,
																			13=Presente con LGV in Richiesta Ingresso e Area Disabilitata,
																			14=Presente con LGV in Ingombro,
																			15=Presente con LGV in Ingombro e Area Disabilitata,
																			16=Presente con LGV Fuori Ingombro e Pallet Estratto,
																			17=Presente con LGV Fuori Ingombro e Pallet Estratto e Area Disabilitata, NOT USED !!!!!!!!!!!
																			99=Errore
																			-1 dato non valido) *)
	F					: INT	:= 0;	(* Forming Pointer - Puntatore tabella formature (1..n=, -1 dato non valido *)
	P					: INT	:= 0;	(* Pack Pointer - Puntatore tabella ELEMENTO (0..n-1=, -1 dato non valido),Numero ELEMENTO successivo da depositare *)
	P_Cava				: Es_PiezasCaballete ;
	
	Code				: INT	:= 0;	(* Codice di Pallettizzazione (0..n=, -1 dato non valido) x lastre, se Magazzino Falde, codice della falda *)
	
	PackPointerModified	: BOOL	:= FALSE;(* Se TRUE, indica che è stata effettuata una modfica sui dati della WA da parte dell' HMI (Settata da HMI e resettata da PLC) *)
	PackPointer			: INT	:= 0;	 (* Rappresenta l'indice del pacco da depositare dopo modfica manuale,cioè con PackPointerModified=TRUE *)

	Slab				: ARRAY[1..MAXFORMINGSLAB] OF TFMachinePalletizer_PlaceElement; (* Struttura Usata per Tracciare Gli Elementi Depositati sulla Workarea *)
	//SlabDimension 		: ARRAY[1..MAXFORMINGSLAB] OF  TFDimensionElement; Ver si hay que añadir
	LGVAttr				: INT := 0;
	BCRead				: ARRAY[1..MAXNUMBARCODE] OF TFMachinePalletizer_BarCode;
	Supporto			: TFMachinePalletizer_Pallet; (* Struttura del supporto presente sulla POSTAZIONE *)
	
	H					: LREAL	:= 0.0; (* (mm) Altezza Reale. Viene calcolata dal PLC dopo ogni prelievo (Vuoti o Falde) o deposito Pallet e durante la pallettizzazione *)
	HPL					: LREAL	:= 0.0; (* (mm) Altezza del pallett utilizzato + altezza layers utilizzati *)
	
	Apprendimento : TFMachinePalletizer_CoordinateApprendimento;(* Apprendimenti nelle varie direzioni *)
	
	
	TransportState : TFMachinePalletizer_WorkAreaTransport_State; (* Stato della WORKAREA quando la Tipologia è TYPOLOGY_OVER_TRANSPORT *)
	
	Slow			: INT	:= 0;		(* Primo Pacco/Lastra in Lenta (0=no, 1=si, -1= non valido) *)
	Taped			: INT	:= 0;		(* Nastratura eseguita. Determina espulsione! (0=non eseguita, 1=eseguita, -1= non valido) *)
	
	Initialize		: BOOL	:= FALSE; 	(* Deposito pallet e falda se prevista ma non continua la pallettizzazione, TRUE= deposita pallet e falda e non continua pallettizzazione, FALSE= Esegue tutto il ciclo regolarmente*)

	
	RefuseLGV       : BOOL	:= FALSE;	(* Abilitazione chiamata LGV a termine pallettizzazione - TRUE= Non chiama LGV quando pallet pieno, FALSE= viene eseguita richiesta LGV *)

	LGV_Req			: INT	:= 0;	(* Richiesta LGV (0=Nop, 1=Richiesta LGV, 2= Consenso Ingresso, -1= non valido) *)
	LGV_GetIn_GetOut: INT	:= 0;	(* Tipo Richiesta LGV  (0=Nop,1=REQ_PRELIEVO_LGV_PIENO,2=REQ_DEPOSITO_LGV_PIENO,3=REQ_PRELIEVO_LGV_VUOTO,4=REQ_DEPOSITO_LGV_VUOTO*)
	//LGV_LetIn		: INT	:= 0;	(* Stato LGV (0=Nop, 1=Richiesta Ingresso, 2=Fine Ingresso, -1= non valido) *)
	//LGV_Footprint	: INT	:= 0;	(* Presenza Ingombro Veicolo (0=Nessun Ingombro, 1=In Ingombro, -1= non valido) *)
	LGV_ReqAbort	: BOOL	:= FALSE; (* Abort chimata LGV *)
	SupportEmpty	: BOOL  := FALSE; (* Se TRUE, con chiamata veicolo attiva significa che l'elemento è vuoto, senza pezzi sopra (lastre o falde) *)
	SupportCentered : BOOL  := FALSE; (* Se TRUE, indica che il supporto è stato centrato *)
	LayerData 		: ST_LayerData; (* Descrizione Falda*)
	SlabData        : ARRAY[1..MAXFORMINGSLAB] OF ST_SlabData;(* Dati delle lastre che servono al supervisore *)
END_STRUCT
END_TYPE

// ---- Data types/Strutture Aggiornate/TFMachinePalletizer_WorkArea.TcDUT
TYPE TFMachinePalletizer_WorkArea :
STRUCT

	Enable			: INT	:= -1;	(* Postazione Abilitata 0=no, 1=si, -1 dato non valido *)
	Typology		: e_Tipo_WorkArea	:= -1;	(* Tipologia 1=Catasta Vuoti, 2=Pallet Singolo, 3=Falda, -1 dato non valido *)
	Typology_Desc   : INT := -1; (* Tipologia Descrittiva della WorkArea*)
	
	Jolly			: INT	:= -1;	(* (Definizione del Codice di Pall... A carico del PLC) (0=no, 1=si, -1= non valido) *)
			
	(* Posizione Assoluta Rispetto a Zero Macchina *)
	X				: LREAL	:= 0.0;	(* READ			- (mm) Quota assoluta di impianto DA ORIGINE *)
	Y				: LREAL	:= 0.0;	(* READ			- (mm) Quota assoluta di impianto DA ORIGINE *)
	Z				: LREAL	:= 0.0;	(* READ			- (mm) Quota assoluta di impianto DA ORIGINE *)
	Rx				: LREAL	:= 0.0;	(* READ			- (°) Angolo di rotazione della postazione Lungo rispetto Asse X *)
	Ry				: LREAL	:= 0.0;	(* READ			- (°) Angolo di rotazione della postazione Lungo rispetto Asse Y *)
	Rz				: LREAL	:= 0.0;	(* READ			- (°) Angolo di rotazione della postazione Lungo rispetto Asse Z *)
	
END_STRUCT
END_TYPE

// ---- Data types/Strutture Aggiornate/TFMachinePalletizer_WorkPickPoint.TcDUT
TYPE TFMachinePalletizer_WorkPickPoint :
STRUCT
	
	Tipologia			: e_Tipo_PickPoint 	:= -1;		(* READ	-	Tipologia del punto di prelievo 
														Per pacchi 	= RIBALTINO;
														Per lastre 	= RULLIERA;
														Per Falde	= MAGAZZIONO_FALDE *)
														
	ID					: INT 	:= -1;		(* READ	-  Identifica il numero del PickPoint *)
	Enable				: INT	:= -1;		(* READ	-  PickPoint Abilitata 0=no, 1=si, -1 dato non valido *)	
(****************************************************** NO LASTRE: ELIMINARE!!! *****************************************************************************************)
	Xv					: LREAL	:= 0.0;		(* READ	- (mm) Quota assoluta di impianto DA ORIGINE - CON RIBALTINO IN VERTICALE - NON USATO PER LASTRE *)
	Yv					: LREAL	:= 0.0;		(* READ	- (mm) Quota assoluta di impianto DA ORIGINE - CON RIBALTINO IN VERTICALE - NON USATO PER LASTRE *)
	Zv					: LREAL	:= 0.0;		(* READ	- (mm) Quota assoluta di impianto DA ORIGINE - CON RIBALTINO IN VERTICALE - NON USATO PER LASTRE *)
	Jv					: LREAL	:= 0.0;		(* READ	- (mm) Quota assoluta di impianto DA ORIGINE - CON RIBALTINO IN VERTICALE - NON USATO PER LASTRE *)
	ZvRaise				: REAL  := 0.0; 	(* READ	- (mm) Quota di salita per uscire dall'ingombro - CON RIBALTINO IN VERTICALE - NON USATO PER LASTRE *)
(***********************************************************************************************************************************************)
	Xh					: LREAL	:= 0.0;		(* READ	- (mm) Quota assoluta di impianto DA ORIGINE - CON RIBALTINO IN ORIZZONTALE - USATO PER LASTRE *)
	Yh					: LREAL	:= 0.0;		(* READ	- (mm) Quota assoluta di impianto DA ORIGINE - CON RIBALTINO IN ORIZZONTALE - USATO PER LASTRE *)
	Zh					: LREAL	:= 0.0;		(* READ	- (mm) Quota assoluta di impianto DA ORIGINE - CON RIBALTINO IN ORIZZONTALE - USATO PER LASTRE *) (*Caso di magazzino falde: è la quota della base di appoggio*)
	Jh					: LREAL	:= 0.0;		(* READ	- (mm) Quota assoluta di impianto DA ORIGINE - CON RIBALTINO IN ORIZZONTALE - USATO PER LASTRE *)
	ZhRaise				: REAL  := 0.0; 	(* READ	- (mm) Quota di salita per uscire dall'ingombro - CON RIBALTINO IN ORIZZONTALE - USATO PER LASTRE *)
	
	Lunghezza			: REAL := 0.0;		(* READ	- (mm) Ingombro in Lunghezza "X" rispetto il suo centro *)
	Larghezza			: REAL := 0.0;		(* READ	- (mm) Ingombro in Larghezza "Y" rispetto il suo centro *)
	Altezza				: REAL := 0.0;		(* READ	- (mm) Ingombro in Altezza "Z" rispetto il suo centro *)
	
	DoLearn_Z			: e_Stato_Apprendimento	:= -1;	(* READ/WRITE 	- Stato apprendimento Direzione Z 0=Disabilitato, 1=Abilitato da Eseguire, 2=Eseguito, -1 dato non valido *)
	Learn_Z				: REAL	:= 0.0;	(* READ			- (mm) Quota inizio Apprendimento Direzione Z *)
	Learned_Z			: LREAL	:= 0.0; (* WRITE		- Quota rilevata durante apprendimento Direzione Z *)
			
END_STRUCT
END_TYPE

// ---- Data types/Strutture Aggiornate/TFMachinePalletizer_WorkArea_VECCHIO.TcDUT
TYPE TFMachinePalletizer_WorkArea_VECCHIO :
STRUCT

	Enable			: INT	:= -1;	(* READ			- Postazione Abilitata 0=no, 1=si, -1 dato non valido *)
	Typology		: e_Tipo_WorkArea	:= -1;	(* READ			- Tipologia 1=Catasta Vuoti, 2=Pallet Singolo, 3=Falda, -1 dato non valido *)
	Typology_Desc	: INT 	:= -1;	(* READ			- Descrizione Dettagliata della Tipologia dell'elmento *)
	Pallet			: INT	:= -1;	(* READ			- Tipo di pallet assegnato (0 = tipo 0, 1 = tipo 1, 2 = tipo 2,  …. , 0 / -1 dato non valido. Usato se Typology=1 *)
	Layer			: INT	:= -1;	(* READ/WRITE	- Tipo di falda dopo il pallet (0 = assente, 1 = tipo 1, 2 = tipo 2,  …. , -1 dato non valido. Usato se Typology=3 *)
	Layer0			: INT 	:= -1;	(* READ/WRITE	- Tipo di falda su cavalletti lato deposito 0° (0 = assente, 1 = tipo 1, 2 = tipo 2,  …. , -1 dato non valido. Usato solo per cavalletti *)
	Layer180		: INT 	:= -1;	(* READ/WRITE	- Tipo di falda su cavalletti lato deposito 180° (0 = assente, 1 = tipo 1, 2 = tipo 2,  …. , -1 dato non valido. Usato solo per cavalletti *)
	Code			: INT	:= -1;	(* READ/WRITE	- Codice di Pallettizzazione (0..n=, -1 dato non valido). Viene estratto dalla Forming se Jolly=1, altrimenti lo si riceve! *)
	Jolly			: INT	:= -1;	(* READ/WRITE	- (Definizione del Codice di Pall... A carico del PLC) (0=no, 1=si, -1= non valido) *)
	
	DoLearn_YDx		: INT	:= -1;	(* READ/WRITE 	- Stato apprendimento Direzione Y verso DX 0=Disabilitato, 1=Abilitato da Eseguire, 2=Eseguito, -1 dato non valido *)
	Learn_YDx		: LREAL	:= 0.0;	(* READ			- (mm) Quota inizio Apprendimento Direzione Y verso DX *)
	Learned_YDx		: LREAL	:= 0.0; (* WRITE		- Quota rilevata durante apprendimento Direzione Y verso DX *)
	DoLearn_YSx		: INT	:= -1;	(* READ/WRITE 	- Stato apprendimento Direzione Y verso SX 0=Disabilitato, 1=Abilitato da Eseguire, 2=Eseguito, -1 dato non valido *)
	Learn_YSx		: LREAL	:= 0.0;	(* READ			- (mm) Quota inizio Apprendimento Direzione Y verso SX *)
	Learned_YSx		: LREAL	:= 0.0; (* WRITE		- Quota rilevata durante apprendimento Direzione Y verso SX *)
	DoLearn_Z		: e_Stato_Apprendimento	:= -1;	(* READ/WRITE 	- Stato apprendimento Direzione Z 0=Disabilitato, 1=Abilitato da Eseguire, 2=Eseguito, -1 dato non valido *)
	Learn_Z			: LREAL	:= 0.0;	(* READ			- (mm) Quota inizio Apprendimento Direzione Z *)
	Learned_Z		: LREAL	:= 0.0; (* WRITE		- Quota rilevata durante apprendimento Direzione Z *)

	Slow			: INT	:= -1;		(* READ			- Primo Pacco/Lastra in Lenta (0=no, 1=si, -1= non valido) *)
	Taped			: INT	:= -1;		(* READ/WRITE	- Nastratura eseguita. Determina espulsione! (0=non eseguita, 1=eseguita, -1= non valido) *)
	RefuseLGV       : BOOL	:= FALSE;	(* READ		- Abilitazione chiamata LGV a termine pallettizzazione - TRUE= Non chiama LGV quando pallet pieno, FALSE= viene eseguita richiesta LGV *)
	Initialize		: BOOL	:= FALSE; 	(* Se TRUE: Blocca la pallettizzazione, mettendo in pausa la postazione *)
	
	X				: LREAL	:= 0.0;	(* READ			- (mm) Quota assoluta di impianto DA ORIGINE *)
	Y				: LREAL	:= 0.0;	(* READ			- (mm) Quota assoluta di impianto DA ORIGINE *)
	Z				: LREAL	:= 0.0;	(* READ			- (mm) Quota assoluta di impianto DA ORIGINE *)
	J				: LREAL	:= 0.0;	(* READ			- (°) Quota assoluta di impianto DA ORIGINE *)
	H				: LREAL	:= 0.0; (* READ/WRITE	- (mm) Altezza Reale. Viene calcolata dal PLC dopo ogni prelievo (Vuoti o Falde) o deposito Pallet e durante la pallettizzazione *)
	HPL				: LREAL	:= 0.0; (* READ/WRITE   - (mm) Altezza del pallett utilizzato + altezza layers utilizzati *)
	
	JPick			: LREAL	:= 0.0;	(* READ			- (°) Quota rotazione EndEffector fase di prelievo *)
	KPick			: LREAL	:= 0.0;	(* READ			- (mm) Quota apertura pinza per prelievo Pacco (usata se la workarea è un magazziono pallet/falde) *)
	JPlace			: LREAL	:= 0.0;	(* READ			- (°) Quota rotazione EndEffector per deposito pallet/falde *)
	
	LGV_Req			: INT	:= 0;	(* READ/WRITE	- Richiesta LGV (0=Nop, 1=Richiesta LGV, 2= Consenso Ingresso, -1= non valido) *)
	LGV_GetIn_GetOut: INT	:= -1;	(* WRITE		- Tipo Richiesta LGV  (0=Nop, 1=Richiesta Prelievo, 2= Richiesta Deposito, -1= non valido) *)	
	LGV_LetIn		: INT	:= -1;	(* READ			- Stato LGV (0=Nop, 1=Richiesta Ingresso, 2=Fine Ingresso, -1= non valido) *)
	LGV_Footprint	: INT	:= -1;	(* READ			- Presenza Ingombro Veicolo (0=Nessun Ingombro, 1=In Ingombro, -1= non valido) *)
	LGV_ReqAbort	: BOOL	:= FALSE; (* READ		- Aborto chimata LGV *)
	
	ProgressiveNr	: UDINT;
	
	IDX_UDCLayer	: INT := 1;	(* Indice che identifica lo strato cassa in lavorazione*)
	
END_STRUCT
END_TYPE

// ---- Data types/Strutture Aggiornate/TFMachinePalletizer_FormingPack.TcDUT
TYPE TFMachinePalletizer_FormingPack :
STRUCT
	
	JP			: INT	:= -1;	(* Tipo di presa (1 = Longitudinale (x), 0 = Trasversale (Y se Verticale, Z se Orizzontale), -1 = dato non valido) *)
	Grip		: INT	:= -1;	(* Tipo di presa (0 = Verticale, 1 = Orizzontale, -1 = dato non valido) *)
	Trajectory	: INT	:= -1;	(* Tipo di percorso (0, 1, 2, 3, …) (-1 dato non valido) *)
	Layer		: INT	:= -1;	(* Tipo di falda dopo il Pacco/Lastra (0 = assente, 1 = tipo 1, 2 = tipo 2,  …. , -1 dato non valido *)
	Nlayer		: INT	:= -1;	(* Numero di falde da depositare dopo il Pacco/Lastra *)
	
	X			: REAL	:= 0.0;	(* (mm) Destination - Coordinata X *)
	Y			: REAL	:= 0.0;	(* (mm) Destination - Coordinata Y *)
	Z			: REAL	:= 0.0;	(* (mm) Destination - Coordinata Z *)
	J			: REAL	:= 0.0;	(* (°)  Destination - Coordinata J *)
	
	AX			: REAL	:= 0.0; (* (mm) Approach X Distance - Distanza Accostamento X *)
	AY			: REAL	:= 0.0; (* (mm) Approach Y Distance - Distanza Accostamento Y *)
	AZ			: REAL	:= 0.0; (* (mm) Approach Z Distance - Distanza Accostamento Z *)
	AJ			: REAL	:= 0.0; (* (°) Approach J Distance - Distanza Accostamento J *)
	
	OffsetDep_0 	: TFMachinePalletizer_OffsetElement; (* OFFSET di deposito, utilizzato per lato 0-90 *)
	OffsetDep_90	: TFMachinePalletizer_OffsetElement; (* OFFSET di deposito, utilizzato per CASSE *)
	OffsetDep_180 	: TFMachinePalletizer_OffsetElement; (* OFFSET di deposito, utilizzato per lato 90-180 *)
	
	UltimoElementoPerUDC	: BOOL	:= FALSE;(*READ - Identifica l'ultimo elemento da depositare in cassa, utilizzato per deposizioni su strati multipli di casse *)

END_STRUCT
END_TYPE

(*
Trajectory :	
 1= standard deposito in diagonale
 2= standard deposito in diagonale specchiato rispetto x
 3=	standard deposito in diagonale specchiato rispetto y
 4= standard deposito in diagonale specchiato rispetto x e y

Layer : quando devo mettere la falda
*)

// ---- Data types/TFDatiDaLineaAPal.TcDUT
TYPE TFDatiDaLineaAPal :
STRUCT

	LastraProntaSuPrelievo 		AT %I* : BOOL;//Lastra pronta sul prelievo i-esimo
	LastraPrelevataDaPrelievo  	AT %Q* : BOOL;//Lastra prelevata da pallettizzatore
	DatiLastraSuPrelievo		AT %I* : TFSlab;
	StatoPrelievo				AT %I* : INT;//Stato rulliera prelievo
	StatoPalettizzatore			AT %Q* : INT;//STtao pallettizzatore
	PinzaInIngombro				AT %Q* : BOOL; //Pinza in ongombro
	
END_STRUCT
END_TYPE

// ---- Data types/TFSlab.TcDUT
TYPE TFSlab :
STRUCT
	
	ID			: UDINT;				(* Unic ID *)
	Code		: UINT;					(* Production Code *)

	X 			: REAL;					(* X dimension *)
	Y 			: REAL;					(* Y dimension *)
	Z 			: REAL;					(* Z dimension *)
	
	StrPos		: ARRAY [1..4] OF REAL;	(* Strapper Position, 	1..8 Straps Position on X *)
	StrDone		: UINT;					(* Strapper Done,  		0=Null, 1..4=N° of Straps Done *)
		
	Centratura	: INT;    (* Stato Centratura*)

	Zone		: INT := e_ElementZone.NULL; //Zona di appartenenza dell'elemento
	Position	: LREAL; (* Posizione in mm sulla cinghia *)
	(* Dati di Classificazione *)
	QualitaPar 	: ARRAY [1..MAXNUMVISIONSYSTEM] OF UINT := [MAXNUMVISIONSYSTEM(0)]; (* Qualità parziale dell'i-esimo Sistema di classificazione (0=UV,1=FlowMaster,..)*)
	TonoPar 	: ARRAY [1..MAXNUMVISIONSYSTEM] OF UINT := [MAXNUMVISIONSYSTEM(0)]; (* Tono parziale dell'i-esimo Sistema di classificazione (0=UV,1=FlowMaster,..)*)		
	StatoLetturaUV : INT := 0; //Indica lo stato della lettura dell'UV (0= Non ancora letto,1= Lettura In Corso,2= Lettura Completata)	
	
	QualitaTot 	: UINT := 0; //Indica la qualità totale data dall'algoritmo impostato
	TonoTot 	: UINT := 0; //Indica il tono totale dato dall'algoritmo impostato
	Calibro		: UINT := 0; //Indica il calibro dato, proveniente direttamente dal sistema calibro-planar

	CreazioneManuale : BOOL;//Indica che l'elemento è stato creato manualmente

END_STRUCT
END_TYPE

// ---- Data types/TF/Aggiornate_20230504/ST_BarcodeReaderReply.TcDUT
//Struttura utilizzata per la lettura dei dati del barcode della Keyence
TYPE ST_BarcodeReaderReply :
STRUCT
	StateComunication 	: UINT;					//Se = 0 comunicazione ok, altrimenti comunicazione interrotta
	Error 				: BOOL;                 //Barcode in errore           
	Busy 				: BOOL;                 //Barcode pronto per nuovo comando
	ReadComplete 		: BOOL;                 //Lettura completata 
	ResultDataAvailable : BOOL;                 //Dato disponibile da Barcode
	GeneralErrorCode 	: UINT;                 //Errore generico da Barcode
	ResultDataSize 		: INT;                  //Dimensione dato letto
	ResultData 			: ARRAY [0..127] OF BYTE; //Dato letto        
	MatchingLevel		: INT;					  //Livello di qualità del dato letto
END_STRUCT
END_TYPE

// ---- Data types/TF/Aggiornate_20230504/ST_BarcodeReaderRequest.TcDUT
//Struttura utilizzata per il comando del barcode della Keyence
TYPE ST_BarcodeReaderRequest :
STRUCT
	ReadRequest 		: BOOL;//Comando di lettura
	ErrorClear 			: BOOL;//Comando azzeramento buffer errori
	ReadCompleteClear 	: BOOL;//Comando azzeramento buffer dati, da mettere a TRUE dopo ogni lettura terminata..
END_STRUCT
END_TYPE

// ---- Data types/TF/Aggiornate_20230504/ST_MachinePalletizerAxeManCmd.TcDUT
TYPE ST_MachinePalletizerAxeManCmd :
STRUCT
	(*  READ	- Home (Ricerca Posizione di Home)  *)
	Home : BOOL := false;
	(*  READ	- Jog +  *)
	JogPos : BOOL := false;
	(*  READ	- Jog -  *)
	JogNeg : BOOL := false;
	(*  READ	- Jog +/- in Fast Speed  *)
	JogFast : BOOL := false;
END_STRUCT
END_TYPE

// ---- Data types/TF/Aggiornate_20230504/ST_MachinePalletizerAxeState.TcDUT
TYPE ST_MachinePalletizerAxeState :
STRUCT
	(*   Actual Position mm  *)
	Position : LREAL := 0;
	(*   Actual Velocity  mm/s  *)
	Velocity : LREAL := 0;
	(*   Actual Torque   *)
	Torque : REAL := 0;
	(*   Error Code   *)
	Error : UDINT := 0;
	(*   TRUE=Power Enable   *)
	PowerActive : BOOL := false;
	(*  Home ok  *)
	Homed : BOOL := false;
END_STRUCT
END_TYPE

// ---- Data types/TF/Aggiornate_20230504/ST_MachinePalletizerMachineState.TcDUT
TYPE ST_MachinePalletizerMachineState :
STRUCT
	(* Comando in esecuzione *)
	Cmd : UDINT;
	(* Stato del comando in esecuzione *)
	CmdCase : UDINT;
	(* Errore generico della Macchina *)
	Error : UDINT;
	(* Errore specifico della Macchina *)
	ErrorExtra : UDINT;
	(* Macchina con potenza attiva *)
	PowerActive : BOOL;
	(* Macchina con Home eseguito *)
	Homed : BOOL;
	(* Macchina in automatico *)
	Auto : BOOL;
	(* Macchina in automatico e con ciclo di lavoro attivo -> sta lavorando *)
	Working : BOOL;
	(* Macchina accesso manuale in area segreta attivo *)
	ManAccesActive : BOOL;
	(* Macchina in Emergenza *)
	EmergencyOK : BOOL;
END_STRUCT
END_TYPE

// ---- Data types/TF/Aggiornate_20230504/ST_MachinePalletizerModuleState.TcDUT
TYPE ST_MachinePalletizerModuleState :
STRUCT
	(* Comando in esecuzione *)
	Cmd : UDINT;
	(* Stato del comando in esecuzione *)
	CmdCase : UDINT;
	(* Errore generico del modulo *)
	Error : UDINT;
	(* Errore specifico del modulo *)
	ErrorExtra : UDINT;
	(* Modulo in Power *)
	PowerActive : BOOL;
	(* Modulo con Home eseguito *)
	Homed : BOOL;
END_STRUCT
END_TYPE

// ---- Data types/TF/Aggiornate_20230504/ST_MachinePalletizerPinzaDeviceState.TcDUT
TYPE ST_MachinePalletizerPinzaDeviceState :
STRUCT
	CilindroApertura 			: TF_CylinderState;//Stato del Cilindro Apertura/chiusura pinza 
	CilindroSbloccoRotazione 	: TF_CylinderState;//Stato del Cilindro Apertura/chiusura pinza 
	AspirazioneFaldaDX 			: TF_CylinderState;//Stato del Cilindro di gestione Aspirazione Falda DX
	AspirazioneFaldaSX 			: TF_CylinderState;//Stato del Cilindro di gestione Aspirazione Falda DX
	AspirazioneDX 				: Ovem_Status;//Stato Vacuostato DX
	AspirazioneSX				: Ovem_Status;//Stato Vacuostato SX
	//CilindroTasteggio 			: TF_CylinderState1;//Stato del Cilindro Tasteggio Pinza 
END_STRUCT
END_TYPE

// ---- Data types/TF/Aggiornate_20230504/ST_MachinePalletizerPinzaStateComplete.TcDUT
TYPE ST_MachinePalletizerPinzaStateComplete :
STRUCT
	(*  Indica che la prolunga DX della pinza è aperta  *)
	LatoDxAperto : BOOL;
	(*  Indica che la prolunga SX della pinza è aperta  *)
	LatoSxAperto : BOOL;
	(*  Indica che la prolunga DX della pinza è chiusa  *)
	LatoDxChiuso : BOOL;
	(*  Indica che la prolunga SX della pinza è chiusa  *)
	LatoSxChiuso : BOOL;
	(*  Indica che sul lato SX ho in presa la piastrella  *)
	LatoSxPiastrellaInPresa : BOOL;
	(*  Indica che sul lato DX ho in presa la piastrella  *)
	LatoDxPiastrellaInPresa : BOOL;
	(*  Indica che sul lato SX ho in presa la FALDA  *)
	LatoSxFaldaInPresa : BOOL;
	(*  Indica che sul lato DX ho in presa la FALDA  *)
	LatoDxFaldaInPresa : BOOL;
	(*  Indica che la Rotazione lungo z è sbloccata  *)
	RotazioneSbloccata : BOOL;
	(*  Indica che la rotazione lungo z è bloccata  *)
	RotazioneBloccata : BOOL;
	(*  Indica che l'elemento è stato prelevato  *)
	ElementoPrelevato : BOOL;
	(*  Indica che il piano è in presa del pezzo  *)
	PianoInPresa : BOOL;
	(*  Stato degli elementi  *)
	ElState : ST_MachinePalletizerPinzaDeviceState;
END_STRUCT
END_TYPE

// ---- Data types/TF/Aggiornate_20230504/ST_MachinePalletizerPinzaVentoseManCmd.TcDUT
TYPE ST_MachinePalletizerPinzaVentoseManCmd:
STRUCT
	(* Attivazione vuoto Ovem DX  *)
	AttivazioneVuotoDX : BOOL;
	(* Attivazione vuoto Ovem SX *)
	AttivazioneVuotoSX : BOOL;
	(* Comandi Ovem *)
	DisattivazioneVuotoDX : BOOL;
	(* Comandi Ove *)
	DisattivazioneVuotoSX : BOOL;
	(* Apertura Pinza *)
	ApriPinza : BOOL;
	(* Apertura Pinza *)
	ChiudiPinza : BOOL;
	(* Sblocco rotazione *)
	SbloccoPinza : BOOL;
	(* Blocco rotazione *)
	BloccoPinza : BOOL;
	(* Attivazione aspirazione Falde DX *)
	AttivazioneVuotoFaldeDX : BOOL;
	(* Disattivazione aspirazione Falde DX *)
	DisattivazioneVuotoFaldeDX : BOOL;
	(* Attivazione aspirazione Falde SX *)
	AttivazioneVuotoFaldeSX : BOOL;
	(* Disattivazione aspirazione Falde SX *)
	DisattivazioneVuotoFaldeSX : BOOL;
	(* Attivazione Tastatori *)
	AttivaTastatori : BOOL;
	(* Disattivazione Tastatori *)
	DisattivaTastatori : BOOL;
	(* Calibrazione OVEM *)
	CalibrazioneOVEM : BOOL;
END_STRUCT
END_TYPE

// ---- Data types/TF/Aggiornate_20230504/ST_StatoPostazioneHMI.TcDUT
TYPE ST_StatoPostazioneHMI :
STRUCT

	Abilitata			: INT; 	 // Abilitazione: 0=Postazione DISABILITATA, 1=Postazione ABILITATA
	TipologiaPostazione	: INT; 	 // Tipologia: 1=Catasta Vuoti, 2=Pallet Singolo, 3=Falda,
	ProgressiveNr 		: INT; //Ad ogni deposito PALLET viene incrementato il suo valore ("ID univoco del pallet depositato")
	
	LGV_Req 			: INT; 	 //Chiamata Navetta: 0=Nessuna Chiamata, 1=Chiamata LGV
	TipologiaSupporto   : INT;
	CodiceLavorazione 	: INT;	 //Codice identificativo di lavorazione 
	
	Stato 				: INT; 	//Stato della Postazione
	CodiceFormatura 	: INT; 	//Codice di Formatura Associata alla postazione
	NPezzi			 	: INT;	//Numero dei pezzi presenti
	
	LGV_Call_EspulsionePieno : BOOL;
	LGV_Call_EspulsioneVuoto : BOOL;
	LGV_Call_RichiestaVuoto : BOOL;
	LGV_Call_RichiestaPieno : BOOL;
	
	LGV_RichiestaIngresso : BOOL;
	LGV_InIngombro : BOOL;
	LGV_OkIngresso : BOOL;	
	
	ID_Supporto 	: INT;//Identificativo supporto
	CampoStringa 	: STRING;//campo per scrittura libera di descrizioni varie esempio: tipo falda

END_STRUCT
END_TYPE

// ---- Data types/TF/Barcode/BarcodeStatus.TcDUT
TYPE BarcodeStatus :
STRUCT
	BarcodeRunMode 	: BOOL; //Barcode in Run Mode
	BarcodeReadRun 	: BOOL; //Barcode in lettura
	ReadDone 		: BOOL; //Lettura terminata
	DataOk 			: BOOL; //Dato valido
	DataMultiple 	: BOOL; //Dato Multiplo Letto
	DataNotRead		: BOOL; //Dato non letto
	ErrorComunication : bool;//Errore comunicazione con barcode/Malfunzionamento dispositivo
END_STRUCT
END_TYPE

// ---- Data types/TF/Barcode/InputDataLogic.TcDUT
TYPE InputDataLogic :
STRUCT

StateETHIP : UINT;
	
ItemSequenceNumber : SINT;
ItemStatus : INT;
ItemDataSize : INT;
LocalPresenceInputBits : SINT;
FailureMask : SINT;
FragmentSequenceNumber : SINT;
FragmentDataSize : INT;
FragmentData : ARRAY [0..127] OF BYTE;

END_STRUCT
END_TYPE

// ---- Data types/TF/Barcode/InputKeyence.TcDUT
TYPE InputKeyence :
STRUCT
	StateComunication	: UINT; //Se = 0 comunicazione ok, altrimenti comunicazione interrotta
	
	Error 				: BOOL;//Barcode in errore
	Busy 				: BOOL;//Barcode pronto per nuovo comando
	
	ReadComplete 		: BOOL;//Barcoda con lettura completa
	ResultDataAvaible 	: BOOL;//Dato disponibile da Barcode
	GeneralErrorCode 	: UINT;//Errore generico da Barcode
	ResultDataSize 		: INT;//Dimensione del dato letto
	
	ResultData 			: ARRAY [0..127] OF BYTE;//Byte di dati letti

	MatchingLevel		: INT; //Percentuale qualità codice letto

END_STRUCT
END_TYPE

// ---- Data types/TF/Barcode/OutputDataLogic.TcDUT
TYPE OutputDataLogic :
STRUCT
	 LastItemSequenceNumberReceived : SINT;
	 RemotePresenceOutputBits : UINT;
	 LastFragmentSequenceNumberReceived : SINT;
END_STRUCT
END_TYPE

// ---- Data types/TF/Barcode/OutputKeyence.TcDUT
TYPE OutputKeyence :
STRUCT
	ReadRequest  		AT %Q* : BOOL;//Comando di lettura
	ErrorClear 	 		AT %Q* : BOOL;//Comando azzeramento buffer errori
	ReadCompleteClear  	AT %Q* : BOOL;//Comando azzeramento buffer dati, da mettere a TRUE dopo ogni lettura terminata..
END_STRUCT
END_TYPE

// ---- Data types/TF/Barcode/StatusDataLogic.TcDUT
TYPE StatusDataLogic :
STRUCT
	BarcodeRunMode 	: BOOL; //Barcode in Run Mode
	BarcodeReadRun 	: BOOL; //Barcode in lettura
	ReadDone 		: BOOL; //Lettura terminata
	DataOk 			: BOOL; //Dato valido
	DataMultiple 	: BOOL; //Dato Multiplo Letto
	DataNotRead		: BOOL; //Dato non letto
	ErrorComunication : bool;//Errore comunicazione con barcode/Malfunzionamento dispositivo
END_STRUCT
END_TYPE

// ---- Data types/TF/Barcode/ST_ManCmdBarcode.TcDUT
TYPE ST_ManCmdBarcode :
STRUCT
	EseguiLettura : BOOL;//Esecuzione ciclo di lettura Barcode
END_STRUCT
END_TYPE

// ---- Data types/TF/Barcode/TFDeviceBCStatus.TcDUT
TYPE TFDeviceBCStatus :
STRUCT

	Device 					: BarcodeStatus;
	DataArray 				: ARRAY[0..127] OF STRING;	//Array di dati
	DataDecode 				: STRING;					//Valore del Dato finale
	UltimeLettureEseguite 	: ARRAY[0..9] OF STRING;	//Memoria Ultime letture eseguite

END_STRUCT
END_TYPE

// ---- Data types/TF/Handling/TFHandlingPack.TcDUT
TYPE TFHandlingPack :
STRUCT
	
	ID			: UDINT;				(* Unic ID *)
	PC			: UINT;					(* Production Code *)
	PP      	: BOOL; 				(* Pack Presence *)

	X 			: REAL;					(* X dimension *)
	Y 			: REAL;					(* Y dimension *)
	Z 			: REAL;					(* Z dimension *)
	
	S1			: UINT;					(* Strapper Number, 	0=No, 1..8=N° of Straps *)
	S1P			: ARRAY [1..8] OF REAL;	(* Strapper Position, 	1..8 Straps Position on X *)
	S1E			: UINT;					(* Strapper Execution,  0=Null, 1..8=N° of Straps in Execution *)
	S1D			: UINT;					(* Strapper Done,  		0=Null, 1..8=N° of Straps Done *)
	S1S			: UINT;					(* Strapper State, 		0=Nop, 1=To Be Worked, 2=Working, 3=Worked *)
	
	S2			: UINT;					(* Strapper Number, 	0=No, 1..8=N° of Straps *)
	S2P			: ARRAY [1..8] OF REAL;	(* Strapper Position, 	1..8 Straps Position on X *)
	S2E			: UINT;					(* Strapper Execution,  0=Null, 1..8=N° of Straps in Execution *)
	S2D			: UINT;					(* Strapper Done,  		0=Null, 1..8=N° of Straps Done *)
	S2S			: UINT;					(* Strapper State, 		0=Nop, 1=To Be Worked, 2=Working, 3=Worked *)
	
	C1 			: UINT;                	(* Coupling Number, 	0=No, 1..8=N° of Packs *)
	C1D			: UINT;					(* Coupling Done,		0=Null, 1..8=N° of Packs Done *)
	
	LB			: BOOL;					(* Label Done,         	TRUE etichetta applicata, FALSE etichetta non applicata *)
	
END_STRUCT
END_TYPE

// ---- Data types/TF/Palletizer/TFMachinePalletizer_AxeState_TF.TcDUT
TYPE TFMachinePalletizer_AxeState_TF :
STRUCT
	
	Position	: LREAL	:= 0.0;	(* Actual Position *)
	Velocity	: LREAL	:= 0.0;	(* Actual Velocity *)
	Torque		: REAL	:= 0.0;	(* Actual Torque *)
	Error		: UDINT	:= 0;	(* Error Code *)
	PowerActive	: BOOL  := FALSE; (* TRUE=Power Enable *)
	
END_STRUCT
END_TYPE

// ---- Data types/TF/Palletizer/TFMachinePalletizer_AxeState_weintek.TcDUT
TYPE TFMachinePalletizer_AxeState_weintek :
STRUCT
	
